ACTION TEST_CASE_1_EXEC:
                        IF vTestCases[0].state = utTestCaseStates.RUNNING THEN
	(*Run the test case*)
	IF assertLessEqual_SINT(vTestCase1_act, vTestCase1_xp) THEN
		vTestCases[0].state := utTestCaseStates.PASSED;
		vTestCases[0].msg := 'Parameter act was less than xp and function returned TRUE -> PASS';
	ELSE
		vTestCases[0].state := utTestCaseStates.FAILED;
		vTestCases[0].msg := 'Parameter act was less than xp and function returned FALSE -> FAIL';
	END_IF
END_IF
                      
END_ACTION

ACTION TEST_CASE_2_SETUP:
                        IF vTestCases[1].state = utTestCaseStates.SETUP THEN
	(*Setup the test case information*)
	vTestCases[1].id := 2;
    vTestCases[1].desc[0] := 'RETURNS TRUE WHEN PARAMETER ACT EQUAL TO XP';
    vTestCases[1].desc[1] := 'Tests if the function returns True if the parameter act is equal to parameter xp';
	vTestCases[1].desc[2] := 'PASS IF: Return value is TRUE';
	
	(*Setup needed variables*)
	vTestCase2_act := REAL_TO_SINT(115.4);
	vTestCase2_xp := REAL_TO_SINT(115.4);
END_IF
                      
END_ACTION

ACTION TEST_CASE_2_EXEC:
                        IF vTestCases[1].state = utTestCaseStates.RUNNING THEN
	(*Run the test case*)
	IF assertLessEqual_SINT(vTestCase2_act, vTestCase2_xp) THEN
		vTestCases[1].state := utTestCaseStates.PASSED;
		vTestCases[1].msg := 'Parameter act was equal to xp and function returned TRUE -> PASS';
	ELSE
		vTestCases[1].state := utTestCaseStates.FAILED;
		vTestCases[1].msg := 'Parameter act was equal to xp and function returned FALSE -> FAIL';
	END_IF
END_IF
                      
END_ACTION

ACTION TEST_CASE_3_SETUP:
                        IF vTestCases[2].state = utTestCaseStates.SETUP THEN
	(*Setup the test case information*)
	vTestCases[2].id := 3;
    vTestCases[2].desc[0] := 'RETURNS FALSE WHEN PARAMETER ACT GREATER THAN XP';
    vTestCases[2].desc[1] := 'Tests if the function returns False if the parameter act is greater than parameter xp';
	vTestCases[2].desc[2] := 'PASS IF: Return value is FALSE';
	
	(*Setup needed variables*)
	vTestCase3_act := REAL_TO_SINT(115.4);
	vTestCase3_xp := REAL_TO_SINT(85.4);
END_IF
                      
END_ACTION

ACTION TEST_CASE_3_EXEC:
                        IF vTestCases[2].state = utTestCaseStates.RUNNING THEN
	(*Run the test case*)
	IF NOT assertLessEqual_SINT(vTestCase3_act, vTestCase3_xp) THEN
		vTestCases[2].state := utTestCaseStates.PASSED;
		vTestCases[2].msg := 'Parameter act was greater than xp and function returned FALSE -> PASS';
	ELSE
		vTestCases[2].state := utTestCaseStates.FAILED;
		vTestCases[2].msg := 'Parameter act was greater than xp and function returned TRUE -> FAIL';
	END_IF
END_IF
                      
END_ACTION
END_PROGRAM

PROGRAM test_assertLess_LDATE
  VAR
    vTestCases : ARRAY[0..20] OF utTestCase;  (* Definition of all test cases for this POU *)
    testRunner : utTestSuite;  (* Test Suite fb instance to run the tests *)
    vRunAll : BOOL;  (* Manual command to run all tests for this POU *)
    vResetAll : BOOL;  (* Manual command to reset all tests for this POU *)
    vTestCase1_act : LDATE;  (* Test data 1 of test case 1 *)
    vTestCase1_xp : LDATE;  (* Test data 2 of test case 1 *)
    vTestCase2_act : LDATE;  (* Test data 1 of test case 2 *)
    vTestCase2_xp : LDATE;  (* Test data 2 of test case 2 *)
  END_VAR

                    (*Run the test cases*)
TEST_CASE_1_SETUP();
TEST_CASE_1_EXEC();

TEST_CASE_2_SETUP();
TEST_CASE_2_EXEC();

(*Instantiate the test runner*)
testRunner(
	Id := 111,
	Name := 'assertLess_LDATE',
    RunTests := GVL.RunAll OR vRunAll,
	ResetTests := GVL.ResetAll OR vResetAll,
	TestCases:=vTestCases);

(*Report the results to the collection global*)
GVL.Results[testRunner.Id] := testRunner.Summary;
                  

ACTION TEST_CASE_2_EXEC:
                        IF vTestCases[1].state = utTestCaseStates.RUNNING THEN
	(*Run the test case*)
	IF NOT assertLess_LDATE(vTestCase2_act, vTestCase2_xp) THEN
		vTestCases[1].state := utTestCaseStates.PASSED;
		vTestCases[1].msg := 'Parameter act was greater than xp and function returned FALSE -> PASS';
	ELSE
		vTestCases[1].state := utTestCaseStates.FAILED;
		vTestCases[1].msg := 'Parameter act was greater than xp and function returned TRUE -> FAIL';
	END_IF
END_IF
                      
END_ACTION

ACTION TEST_CASE_1_SETUP:
                        IF vTestCases[0].state = utTestCaseStates.SETUP THEN
	(*Setup the test case information*)
	vTestCases[0].id := 1;
	vTestCases[0].desc[0] := 'RETURNS TRUE WHEN PARAMETER ACT LESS THAN XP';
    vTestCases[0].desc[1] := 'Tests if the function returns True if the parameter act is less than parameter xp';
	vTestCases[0].desc[2] := 'PASS IF: Return value is TRUE';
	
	(*Setup needed variables*)
	vTestCase1_act := REAL_TO_LDATE(85.4);
	vTestCase1_xp := REAL_TO_LDATE(115.4);
END_IF
                      
END_ACTION

ACTION TEST_CASE_1_EXEC:
                        IF vTestCases[0].state = utTestCaseStates.RUNNING THEN
	(*Run the test case*)
	IF assertLess_LDATE(vTestCase1_act, vTestCase1_xp) THEN
		vTestCases[0].state := utTestCaseStates.PASSED;
		vTestCases[0].msg := 'Parameter act was less than xp and function returned TRUE -> PASS';
	ELSE
		vTestCases[0].state := utTestCaseStates.FAILED;
		vTestCases[0].msg := 'Parameter act was less than xp and function returned FALSE -> FAIL';
	END_IF
END_IF
                      
END_ACTION

ACTION TEST_CASE_2_SETUP:
                        IF vTestCases[1].state = utTestCaseStates.SETUP THEN
	(*Setup the test case information*)
	vTestCases[1].id := 2;
    vTestCases[1].desc[0] := 'RETURNS FALSE WHEN PARAMETER ACT GREATER THAN XP';
    vTestCases[1].desc[1] := 'Tests if the function returns False if the parameter act is greater than parameter xp';
	vTestCases[1].desc[2] := 'PASS IF: Return value is FALSE';
	
	(*Setup needed variables*)
	vTestCase2_act := REAL_TO_LDATE(115.4);
	vTestCase2_xp := REAL_TO_LDATE(85.4);
END_IF
                      
END_ACTION
END_PROGRAM

PROGRAM test_assertLess_ULINT
  VAR
    vTestCases : ARRAY[0..20] OF utTestCase;  (* Definition of all test cases for this POU *)
    testRunner : utTestSuite;  (* Test Suite fb instance to run the tests *)
    vRunAll : BOOL;  (* Manual command to run all tests for this POU *)
    vResetAll : BOOL;  (* Manual command to reset all tests for this POU *)
    vTestCase1_act : ULINT;  (* Test data 1 of test case 1 *)
    vTestCase1_xp : ULINT;  (* Test data 2 of test case 1 *)
    vTestCase2_act : ULINT;  (* Test data 1 of test case 2 *)
    vTestCase2_xp : ULINT;  (* Test data 2 of test case 2 *)
  END_VAR

                    (*Run the test cases*)
TEST_CASE_1_SETUP();
TEST_CASE_1_EXEC();

TEST_CASE_2_SETUP();
TEST_CASE_2_EXEC();

(*Instantiate the test runner*)
testRunner(
	Id := 105,
	Name := 'assertLess_ULINT',
    RunTests := GVL.RunAll OR vRunAll,
	ResetTests := GVL.ResetAll OR vResetAll,
	TestCases:=vTestCases);

(*Report the results to the collection global*)
GVL.Results[testRunner.Id] := testRunner.Summary;
                  

ACTION TEST_CASE_1_SETUP:
                        IF vTestCases[0].state = utTestCaseStates.SETUP THEN
	(*Setup the test case information*)
	vTestCases[0].id := 1;
	vTestCases[0].desc[0] := 'RETURNS TRUE WHEN PARAMETER ACT LESS THAN XP';
    vTestCases[0].desc[1] := 'Tests if the function returns True if the parameter act is less than parameter xp';
	vTestCases[0].desc[2] := 'PASS IF: Return value is TRUE';
	
	(*Setup needed variables*)
	vTestCase1_act := REAL_TO_ULINT(85.4);
	vTestCase1_xp := REAL_TO_ULINT(115.4);
END_IF
                      
END_ACTION

ACTION TEST_CASE_1_EXEC:
                        IF vTestCases[0].state = utTestCaseStates.RUNNING THEN
	(*Run the test case*)
	IF assertLess_ULINT(vTestCase1_act, vTestCase1_xp) THEN
		vTestCases[0].state := utTestCaseStates.PASSED;
		vTestCases[0].msg := 'Parameter act was less than xp and function returned TRUE -> PASS';
	ELSE
		vTestCases[0].state := utTestCaseStates.FAILED;
		vTestCases[0].msg := 'Parameter act was less than xp and function returned FALSE -> FAIL';
	END_IF
END_IF
                      
END_ACTION

ACTION TEST_CASE_2_SETUP:
                        IF vTestCases[1].state = utTestCaseStates.SETUP THEN
	(*Setup the test case information*)
	vTestCases[1].id := 2;
    vTestCases[1].desc[0] := 'RETURNS FALSE WHEN PARAMETER ACT GREATER THAN XP';
    vTestCases[1].desc[1] := 'Tests if the function returns False if the parameter act is greater than parameter xp';
	vTestCases[1].desc[2] := 'PASS IF: Return value is FALSE';
	
	(*Setup needed variables*)
	vTestCase2_act := REAL_TO_ULINT(115.4);
	vTestCase2_xp := REAL_TO_ULINT(85.4);
END_IF
                      
END_ACTION

ACTION TEST_CASE_2_EXEC:
                        IF vTestCases[1].state = utTestCaseStates.RUNNING THEN
	(*Run the test case*)
	IF NOT assertLess_ULINT(vTestCase2_act, vTestCase2_xp) THEN
		vTestCases[1].state := utTestCaseStates.PASSED;
		vTestCases[1].msg := 'Parameter act was greater than xp and function returned FALSE -> PASS';
	ELSE
		vTestCases[1].state := utTestCaseStates.FAILED;
		vTestCases[1].msg := 'Parameter act was greater than xp and function returned TRUE -> FAIL';
	END_IF
END_IF
                      
END_ACTION
END_PROGRAM

PROGRAM test_assertLess_REAL
  VAR
    vTestCases : ARRAY[0..20] OF utTestCase;  (* Definition of all test cases for this POU *)
    testRunner : utTestSuite;  (* Test Suite fb instance to run the tests *)
    vRunAll : BOOL;  (* Manual command to run all tests for this POU *)
    vResetAll : BOOL;  (* Manual command to reset all tests for this POU *)
    vTestCase1_act : REAL;  (* Test data 1 of test case 1 *)
    vTestCase1_xp : REAL;  (* Test data 2 of test case 1 *)
    vTestCase2_act : REAL;  (* Test data 1 of test case 2 *)
    vTestCase2_xp : REAL;  (* Test data 2 of test case 2 *)
  END_VAR

                    (*Run the test cases*)
TEST_CASE_1_SETUP();
TEST_CASE_1_EXEC();

TEST_CASE_2_SETUP();
TEST_CASE_2_EXEC();

(*Instantiate the test runner*)
testRunner(
	Id := 106,
	Name := 'assertLess_REAL',
    RunTests := GVL.RunAll OR vRunAll,
	ResetTests := GVL.ResetAll OR vResetAll,
	TestCases:=vTestCases);

(*Report the results to the collection global*)
GVL.Results[testRunner.Id] := testRunner.Summary;
                  

ACTION TEST_CASE_1_SETUP:
                        IF vTestCases[0].state = utTestCaseStates.SETUP THEN
	(*Setup the test case information*)
	vTestCases[0].id := 1;
	vTestCases[0].desc[0] := 'RETURNS TRUE WHEN PARAMETER ACT LESS THAN XP';
    vTestCases[0].desc[1] := 'Tests if the function returns True if the parameter act is less than parameter xp';
	vTestCases[0].desc[2] := 'PASS IF: Return value is TRUE';
	
	(*Setup needed variables*)
	vTestCase1_act := 85.4;
	vTestCase1_xp := 115.4;
END_IF
                      
END_ACTION

ACTION TEST_CASE_1_EXEC:
                        IF vTestCases[0].state = utTestCaseStates.RUNNING THEN
	(*Run the test case*)
	IF assertLess_REAL(vTestCase1_act, vTestCase1_xp) THEN
		vTestCases[0].state := utTestCaseStates.PASSED;
		vTestCases[0].msg := 'Parameter act was less than xp and function returned TRUE -> PASS';
	ELSE
		vTestCases[0].state := utTestCaseStates.FAILED;
		vTestCases[0].msg := 'Parameter act was less than xp and function returned FALSE -> FAIL';
	END_IF
END_IF
                      
END_ACTION

ACTION TEST_CASE_2_SETUP:
                        IF vTestCases[1].state = utTestCaseStates.SETUP THEN
	(*Setup the test case information*)
	vTestCases[1].id := 2;
    vTestCases[1].desc[0] := 'RETURNS FALSE WHEN PARAMETER ACT GREATER THAN XP';
    vTestCases[1].desc[1] := 'Tests if the function returns False if the parameter act is greater than parameter xp';
	vTestCases[1].desc[2] := 'PASS IF: Return value is FALSE';
	
	(*Setup needed variables*)
	vTestCase2_act := 115.4;
	vTestCase2_xp := 85.4;
END_IF
                      
END_ACTION

ACTION TEST_CASE_2_EXEC:
                        IF vTestCases[1].state = utTestCaseStates.RUNNING THEN
	(*Run the test case*)
	IF NOT assertLess_REAL(vTestCase2_act, vTestCase2_xp) THEN
		vTestCases[1].state := utTestCaseStates.PASSED;
		vTestCases[1].msg := 'Parameter act was greater than xp and function returned FALSE -> PASS';
	ELSE
		vTestCases[1].state := utTestCaseStates.FAILED;
		vTestCases[1].msg := 'Parameter act was greater than xp and function returned TRUE -> FAIL';
	END_IF
END_IF
                      
END_ACTION
END_PROGRAM

PROGRAM test_assertLess_TIME_OF_DAY
  VAR
    vTestCases : ARRAY[0..20] OF utTestCase;  (* Definition of all test cases for this POU *)
    testRunner : utTestSuite;  (* Test Suite fb instance to run the tests *)
    vRunAll : BOOL;  (* Manual command to run all tests for this POU *)
    vResetAll : BOOL;  (* Manual command to reset all tests for this POU *)
    vTestCase1_act : TOD;  (* Test data 1 of test case 1 *)
    vTestCase1_xp : TOD;  (* Test data 2 of test case 1 *)
    vTestCase2_act : TOD;  (* Test data 1 of test case 2 *)
    vTestCase2_xp : TOD;  (* Test data 2 of test case 2 *)
  END_VAR

                    (*Run the test cases*)
TEST_CASE_1_SETUP();
TEST_CASE_1_EXEC();

TEST_CASE_2_SETUP();
TEST_CASE_2_EXEC();

(*Instantiate the test runner*)
testRunner(
	Id := 114,
	Name := 'assertLess_TIME_OF_DAY',
    RunTests := GVL.RunAll OR vRunAll,
	ResetTests := GVL.ResetAll OR vResetAll,
	TestCases:=vTestCases);

(*Report the results to the collection global*)
GVL.Results[testRunner.Id] := testRunner.Summary;
                  

ACTION TEST_CASE_2_SETUP:
                        IF vTestCases[1].state = utTestCaseStates.SETUP THEN
	(*Setup the test case information*)
	vTestCases[1].id := 2;
    vTestCases[1].desc[0] := 'RETURNS FALSE WHEN PARAMETER ACT GREATER THAN XP';
    vTestCases[1].desc[1] := 'Tests if the function returns False if the parameter act is greater than parameter xp';
	vTestCases[1].desc[2] := 'PASS IF: Return value is FALSE';
	
	(*Setup needed variables*)
	vTestCase2_act := REAL_TO_TOD(115.4);
	vTestCase2_xp := REAL_TO_TOD(85.4);
END_IF
                      
END_ACTION

ACTION TEST_CASE_1_SETUP:
                        IF vTestCases[0].state = utTestCaseStates.SETUP THEN
	(*Setup the test case information*)
	vTestCases[0].id := 1;
	vTestCases[0].desc[0] := 'RETURNS TRUE WHEN PARAMETER ACT LESS THAN XP';
    vTestCases[0].desc[1] := 'Tests if the function returns True if the parameter act is less than parameter xp';
	vTestCases[0].desc[2] := 'PASS IF: Return value is TRUE';
	
	(*Setup needed variables*)
	vTestCase1_act := REAL_TO_TOD(85.4);
	vTestCase1_xp := REAL_TO_TOD(115.4);
END_IF
                      
END_ACTION

ACTION TEST_CASE_1_EXEC:
                        IF vTestCases[0].state = utTestCaseStates.RUNNING THEN
	(*Run the test case*)
	IF assertLess_TIME_OF_DAY(vTestCase1_act, vTestCase1_xp) THEN
		vTestCases[0].state := utTestCaseStates.PASSED;
		vTestCases[0].msg := 'Parameter act was less than xp and function returned TRUE -> PASS';
	ELSE
		vTestCases[0].state := utTestCaseStates.FAILED;
		vTestCases[0].msg := 'Parameter act was less than xp and function returned FALSE -> FAIL';
	END_IF
END_IF
                      
END_ACTION

ACTION TEST_CASE_2_EXEC:
                        IF vTestCases[1].state = utTestCaseStates.RUNNING THEN
	(*Run the test case*)
	IF NOT assertLess_TIME_OF_DAY(vTestCase2_act, vTestCase2_xp) THEN
		vTestCases[1].state := utTestCaseStates.PASSED;
		vTestCases[1].msg := 'Parameter act was greater than xp and function returned FALSE -> PASS';
	ELSE
		vTestCases[1].state := utTestCaseStates.FAILED;
		vTestCases[1].msg := 'Parameter act was greater than xp and function returned TRUE -> FAIL';
	END_IF
END_IF
                      
END_ACTION
END_PROGRAM

PROGRAM test_assertLess_LREAL
  VAR
    vTestCases : ARRAY[0..20] OF utTestCase;  (* Definition of all test cases for this POU *)
    testRunner : utTestSuite;  (* Test Suite fb instance to run the tests *)
    vRunAll : BOOL;  (* Manual command to run all tests for this POU *)
    vResetAll : BOOL;  (* Manual command to reset all tests for this POU *)
    vTestCase1_act : LREAL;  (* Test data 1 of test case 1 *)
    vTestCase1_xp : LREAL;  (* Test data 2 of test case 1 *)
    vTestCase2_act : LREAL;  (* Test data 1 of test case 2 *)
    vTestCase2_xp : LREAL;  (* Test data 2 of test case 2 *)
  END_VAR

                    (*Run the test cases*)
TEST_CASE_1_SETUP();
TEST_CASE_1_EXEC();

TEST_CASE_2_SETUP();
TEST_CASE_2_EXEC();

(*Instantiate the test runner*)
testRunner(
	Id := 107,
	Name := 'assertLess_LREAL',
    RunTests := GVL.RunAll OR vRunAll,
	ResetTests := GVL.ResetAll OR vResetAll,
	TestCases:=vTestCases);

(*Report the results to the collection global*)
GVL.Results[testRunner.Id] := testRunner.Summary;
                  

ACTION TEST_CASE_2_SETUP:
                        IF vTestCases[1].state = utTestCaseStates.SETUP THEN
	(*Setup the test case information*)
	vTestCases[1].id := 2;
    vTestCases[1].desc[0] := 'RETURNS FALSE WHEN PARAMETER ACT GREATER THAN XP';
    vTestCases[1].desc[1] := 'Tests if the function returns False if the parameter act is greater than parameter xp';
	vTestCases[1].desc[2] := 'PASS IF: Return value is FALSE';
	
	(*Setup needed variables*)
	vTestCase2_act := REAL_TO_LREAL(115.4);
	vTestCase2_xp := REAL_TO_LREAL(85.4);
END_IF
                      
END_ACTION

ACTION TEST_CASE_1_SETUP:
                        IF vTestCases[0].state = utTestCaseStates.SETUP THEN
	(*Setup the test case information*)
	vTestCases[0].id := 1;
	vTestCases[0].desc[0] := 'RETURNS TRUE WHEN PARAMETER ACT LESS THAN XP';
    vTestCases[0].desc[1] := 'Tests if the function returns True if the parameter act is less than parameter xp';
	vTestCases[0].desc[2] := 'PASS IF: Return value is TRUE';
	
	(*Setup needed variables*)
	vTestCase1_act := REAL_TO_LREAL(85.4);
	vTestCase1_xp := REAL_TO_LREAL(115.4);
END_IF
                      
END_ACTION

ACTION TEST_CASE_1_EXEC:
                        IF vTestCases[0].state = utTestCaseStates.RUNNING THEN
	(*Run the test case*)
	IF assertLess_LREAL(vTestCase1_act, vTestCase1_xp) THEN
		vTestCases[0].state := utTestCaseStates.PASSED;
		vTestCases[0].msg := 'Parameter act was less than xp and function returned TRUE -> PASS';
	ELSE
		vTestCases[0].state := utTestCaseStates.FAILED;
		vTestCases[0].msg := 'Parameter act was less than xp and function returned FALSE -> FAIL';
	END_IF
END_IF
                      
END_ACTION

ACTION TEST_CASE_2_EXEC:
                        IF vTestCases[1].state = utTestCaseStates.RUNNING THEN
	(*Run the test case*)
	IF NOT assertLess_LREAL(vTestCase2_act, vTestCase2_xp) THEN
		vTestCases[1].state := utTestCaseStates.PASSED;
		vTestCases[1].msg := 'Parameter act was greater than xp and function returned FALSE -> PASS';
	ELSE
		vTestCases[1].state := utTestCaseStates.FAILED;
		vTestCases[1].msg := 'Parameter act was greater than xp and function returned TRUE -> FAIL';
	END_IF
END_IF
                      
END_ACTION
END_PROGRAM

PROGRAM test_assertLess_BYTE
  VAR
    vTestCases : ARRAY[0..20] OF utTestCase;  (* Definition of all test cases for this POU *)
    testRunner : utTestSuite;  (* Test Suite fb instance to run the tests *)
    vRunAll : BOOL;  (* Manual command to run all tests for this POU *)
    vResetAll : BOOL;  (* Manual command to reset all tests for this POU *)
    vTestCase1_act : BYTE;  (* Test data 1 of test case 1 *)
    vTestCase1_xp : BYTE;  (* Test data 2 of test case 1 *)
    vTestCase2_act : BYTE;  (* Test data 1 of test case 2 *)
    vTestCase2_xp : BYTE;  (* Test data 2 of test case 2 *)
  END_VAR

                    (*Run the test cases*)
TEST_CASE_1_SETUP();
TEST_CASE_1_EXEC();

TEST_CASE_2_SETUP();
TEST_CASE_2_EXEC();

(*Instantiate the test runner*)
testRunner(
	Id := 94,
	Name := 'assertLess_BYTE',
    RunTests := GVL.RunAll OR vRunAll,
	ResetTests := GVL.ResetAll OR vResetAll,
	TestCases:=vTestCases);

(*Report the results to the collection global*)
GVL.Results[testRunner.Id] := testRunner.Summary;
                  

ACTION TEST_CASE_1_SETUP:
                        IF vTestCases[0].state = utTestCaseStates.SETUP THEN
	(*Setup the test case information*)
	vTestCases[0].id := 1;
	vTestCases[0].desc[0] := 'RETURNS TRUE WHEN PARAMETER ACT LESS THAN XP';
    vTestCases[0].desc[1] := 'Tests if the function returns True if the parameter act is less than parameter xp';
	vTestCases[0].desc[2] := 'PASS IF: Return value is TRUE';
	
	(*Setup needed variables*)
	vTestCase1_act := REAL_TO_BYTE(85.4);
	vTestCase1_xp := REAL_TO_BYTE(115.4);
END_IF
                      
END_ACTION

ACTION TEST_CASE_1_EXEC:
                        IF vTestCases[0].state = utTestCaseStates.RUNNING THEN
	(*Run the test case*)
	IF assertLess_BYTE(vTestCase1_act, vTestCase1_xp) THEN
		vTestCases[0].state := utTestCaseStates.PASSED;
		vTestCases[0].msg := 'Parameter act was less than xp and function returned TRUE -> PASS';
	ELSE
		vTestCases[0].state := utTestCaseStates.FAILED;
		vTestCases[0].msg := 'Parameter act was less than xp and function returned FALSE -> FAIL';
	END_IF
END_IF
                      
END_ACTION

ACTION TEST_CASE_2_SETUP:
                        IF vTestCases[1].state = utTestCaseStates.SETUP THEN
	(*Setup the test case information*)
	vTestCases[1].id := 2;
    vTestCases[1].desc[0] := 'RETURNS FALSE WHEN PARAMETER ACT GREATER THAN XP';
    vTestCases[1].desc[1] := 'Tests if the function returns False if the parameter act is greater than parameter xp';
	vTestCases[1].desc[2] := 'PASS IF: Return value is FALSE';
	
	(*Setup needed variables*)
	vTestCase2_act := REAL_TO_BYTE(115.4);
	vTestCase2_xp := REAL_TO_BYTE(85.4);
END_IF
                      
END_ACTION

ACTION TEST_CASE_2_EXEC:
                        IF vTestCases[1].state = utTestCaseStates.RUNNING THEN
	(*Run the test case*)
	IF NOT assertLess_BYTE(vTestCase2_act, vTestCase2_xp) THEN
		vTestCases[1].state := utTestCaseStates.PASSED;
		vTestCases[1].msg := 'Parameter act was greater than xp and function returned FALSE -> PASS';
	ELSE
		vTestCases[1].state := utTestCaseStates.FAILED;
		vTestCases[1].msg := 'Parameter act was greater than xp and function returned TRUE -> FAIL';
	END_IF
END_IF
                      
END_ACTION
END_PROGRAM

PROGRAM test_assertLess_UINT
  VAR
    vTestCases : ARRAY[0..20] OF utTestCase;  (* Definition of all test cases for this POU *)
    testRunner : utTestSuite;  (* Test Suite fb instance to run the tests *)
    vRunAll : BOOL;  (* Manual command to run all tests for this POU *)
    vResetAll : BOOL;  (* Manual command to reset all tests for this POU *)
    vTestCase1_act : UINT;  (* Test data 1 of test case 1 *)
    vTestCase1_xp : UINT;  (* Test data 2 of test case 1 *)
    vTestCase2_act : UINT;  (* Test data 1 of test case 2 *)
    vTestCase2_xp : UINT;  (* Test data 2 of test case 2 *)
  END_VAR

                    (*Run the test cases*)
TEST_CASE_1_SETUP();
TEST_CASE_1_EXEC();

TEST_CASE_2_SETUP();
TEST_CASE_2_EXEC();

(*Instantiate the test runner*)
testRunner(
	Id := 101,
	Name := 'assertLess_UINT',
    RunTests := GVL.RunAll OR vRunAll,
	ResetTests := GVL.ResetAll OR vResetAll,
	TestCases:=vTestCases);

(*Report the results to the collection global*)
GVL.Results[testRunner.Id] := testRunner.Summary;
                  

ACTION TEST_CASE_1_SETUP:
                        IF vTestCases[0].state = utTestCaseStates.SETUP THEN
	(*Setup the test case information*)
	vTestCases[0].id := 1;
	vTestCases[0].desc[0] := 'RETURNS TRUE WHEN PARAMETER ACT LESS THAN XP';
    vTestCases[0].desc[1] := 'Tests if the function returns True if the parameter act is less than parameter xp';
	vTestCases[0].desc[2] := 'PASS IF: Return value is TRUE';
	
	(*Setup needed variables*)
	vTestCase1_act := REAL_TO_UINT(85.4);
	vTestCase1_xp := REAL_TO_UINT(115.4);
END_IF
                      
END_ACTION

ACTION TEST_CASE_1_EXEC:
                        IF vTestCases[0].state = utTestCaseStates.RUNNING THEN
	(*Run the test case*)
	IF assertLess_UINT(vTestCase1_act, vTestCase1_xp) THEN
		vTestCases[0].state := utTestCaseStates.PASSED;
		vTestCases[0].msg := 'Parameter act was less than xp and function returned TRUE -> PASS';
	ELSE
		vTestCases[0].state := utTestCaseStates.FAILED;
		vTestCases[0].msg := 'Parameter act was less than xp and function returned FALSE -> FAIL';
	END_IF
END_IF
                      
END_ACTION

ACTION TEST_CASE_2_SETUP:
                        IF vTestCases[1].state = utTestCaseStates.SETUP THEN
	(*Setup the test case information*)
	vTestCases[1].id := 2;
    vTestCases[1].desc[0] := 'RETURNS FALSE WHEN PARAMETER ACT GREATER THAN XP';
    vTestCases[1].desc[1] := 'Tests if the function returns False if the parameter act is greater than parameter xp';
	vTestCases[1].desc[2] := 'PASS IF: Return value is FALSE';
	
	(*Setup needed variables*)
	vTestCase2_act := REAL_TO_UINT(115.4);
	vTestCase2_xp := REAL_TO_UINT(85.4);
END_IF
                      
END_ACTION

ACTION TEST_CASE_2_EXEC:
                        IF vTestCases[1].state = utTestCaseStates.RUNNING THEN
	(*Run the test case*)
	IF NOT assertLess_UINT(vTestCase2_act, vTestCase2_xp) THEN
		vTestCases[1].state := utTestCaseStates.PASSED;
		vTestCases[1].msg := 'Parameter act was greater than xp and function returned FALSE -> PASS';
	ELSE
		vTestCases[1].state := utTestCaseStates.FAILED;
		vTestCases[1].msg := 'Parameter act was greater than xp and function returned TRUE -> FAIL';
	END_IF
END_IF
                      
END_ACTION
END_PROGRAM

PROGRAM test_assertLess_DWORD
  VAR
    vTestCases : ARRAY[0..20] OF utTestCase;  (* Definition of all test cases for this POU *)
    testRunner : utTestSuite;  (* Test Suite fb instance to run the tests *)
    vRunAll : BOOL;  (* Manual command to run all tests for this POU *)
    vResetAll : BOOL;  (* Manual command to reset all tests for this POU *)
    vTestCase1_act : DWORD;  (* Test data 1 of test case 1 *)
    vTestCase1_xp : DWORD;  (* Test data 2 of test case 1 *)
    vTestCase2_act : DWORD;  (* Test data 1 of test case 2 *)
    vTestCase2_xp : DWORD;  (* Test data 2 of test case 2 *)
  END_VAR

                    (*Run the test cases*)
TEST_CASE_1_SETUP();
TEST_CASE_1_EXEC();

TEST_CASE_2_SETUP();
TEST_CASE_2_EXEC();

(*Instantiate the test runner*)
testRunner(
	Id := 96,
	Name := 'assertLess_DWORD',
    RunTests := GVL.RunAll OR vRunAll,
	ResetTests := GVL.ResetAll OR vResetAll,
	TestCases:=vTestCases);

(*Report the results to the collection global*)
GVL.Results[testRunner.Id] := testRunner.Summary;
                  

ACTION TEST_CASE_1_EXEC:
                        IF vTestCases[0].state = utTestCaseStates.RUNNING THEN
	(*Run the test case*)
	IF assertLess_DWORD(vTestCase1_act, vTestCase1_xp) THEN
		vTestCases[0].state := utTestCaseStates.PASSED;
		vTestCases[0].msg := 'Parameter act was less than xp and function returned TRUE -> PASS';
	ELSE
		vTestCases[0].state := utTestCaseStates.FAILED;
		vTestCases[0].msg := 'Parameter act was less than xp and function returned FALSE -> FAIL';
	END_IF
END_IF
                      
END_ACTION

ACTION TEST_CASE_2_SETUP:
                        IF vTestCases[1].state = utTestCaseStates.SETUP THEN
	(*Setup the test case information*)
	vTestCases[1].id := 2;
    vTestCases[1].desc[0] := 'RETURNS FALSE WHEN PARAMETER ACT GREATER THAN XP';
    vTestCases[1].desc[1] := 'Tests if the function returns False if the parameter act is greater than parameter xp';
	vTestCases[1].desc[2] := 'PASS IF: Return value is FALSE';
	
	(*Setup needed variables*)
	vTestCase2_act := REAL_TO_DWORD(115.4);
	vTestCase2_xp := REAL_TO_DWORD(85.4);
END_IF
                      
END_ACTION

ACTION TEST_CASE_2_EXEC:
                        IF vTestCases[1].state = utTestCaseStates.RUNNING THEN
	(*Run the test case*)
	IF NOT assertLess_DWORD(vTestCase2_act, vTestCase2_xp) THEN
		vTestCases[1].state := utTestCaseStates.PASSED;
		vTestCases[1].msg := 'Parameter act was greater than xp and function returned FALSE -> PASS';
	ELSE
		vTestCases[1].state := utTestCaseStates.FAILED;
		vTestCases[1].msg := 'Parameter act was greater than xp and function returned TRUE -> FAIL';
	END_IF
END_IF
                      
END_ACTION

ACTION TEST_CASE_1_SETUP:
                        IF vTestCases[0].state = utTestCaseStates.SETUP THEN
	(*Setup the test case information*)
	vTestCases[0].id := 1;
	vTestCases[0].desc[0] := 'RETURNS TRUE WHEN PARAMETER ACT LESS THAN XP';
    vTestCases[0].desc[1] := 'Tests if the function returns True if the parameter act is less than parameter xp';
	vTestCases[0].desc[2] := 'PASS IF: Return value is TRUE';
	
	(*Setup needed variables*)
	vTestCase1_act := REAL_TO_DWORD(85.4);
	vTestCase1_xp := REAL_TO_DWORD(115.4);
END_IF
                      
END_ACTION
END_PROGRAM

PROGRAM test_assertLess_UDINT
  VAR
    vTestCases : ARRAY[0..20] OF utTestCase;  (* Definition of all test cases for this POU *)
    testRunner : utTestSuite;  (* Test Suite fb instance to run the tests *)
    vRunAll : BOOL;  (* Manual command to run all tests for this POU *)
    vResetAll : BOOL;  (* Manual command to reset all tests for this POU *)
    vTestCase1_act : UDINT;  (* Test data 1 of test case 1 *)
    vTestCase1_xp : UDINT;  (* Test data 2 of test case 1 *)
    vTestCase2_act : UDINT;  (* Test data 1 of test case 2 *)
    vTestCase2_xp : UDINT;  (* Test data 2 of test case 2 *)
  END_VAR

                    (*Run the test cases*)
TEST_CASE_1_SETUP();
TEST_CASE_1_EXEC();

TEST_CASE_2_SETUP();
TEST_CASE_2_EXEC();

(*Instantiate the test runner*)
testRunner(
	Id := 103,
	Name := 'assertLess_UDINT',
    RunTests := GVL.RunAll OR vRunAll,
	ResetTests := GVL.ResetAll OR vResetAll,
	TestCases:=vTestCases);

(*Report the results to the collection global*)
GVL.Results[testRunner.Id] := testRunner.Summary;
                  

ACTION TEST_CASE_1_EXEC:
                        IF vTestCases[0].state = utTestCaseStates.RUNNING THEN
	(*Run the test case*)
	IF assertLess_UDINT(vTestCase1_act, vTestCase1_xp) THEN
		vTestCases[0].state := utTestCaseStates.PASSED;
		vTestCases[0].msg := 'Parameter act was less than xp and function returned TRUE -> PASS';
	ELSE
		vTestCases[0].state := utTestCaseStates.FAILED;
		vTestCases[0].msg := 'Parameter act was less than xp and function returned FALSE -> FAIL';
	END_IF
END_IF
                      
END_ACTION

ACTION TEST_CASE_2_SETUP:
                        IF vTestCases[1].state = utTestCaseStates.SETUP THEN
	(*Setup the test case information*)
	vTestCases[1].id := 2;
    vTestCases[1].desc[0] := 'RETURNS FALSE WHEN PARAMETER ACT GREATER THAN XP';
    vTestCases[1].desc[1] := 'Tests if the function returns False if the parameter act is greater than parameter xp';
	vTestCases[1].desc[2] := 'PASS IF: Return value is FALSE';
	
	(*Setup needed variables*)
	vTestCase2_act := REAL_TO_UDINT(115.4);
	vTestCase2_xp := REAL_TO_UDINT(85.4);
END_IF
                      
END_ACTION

ACTION TEST_CASE_2_EXEC:
                        IF vTestCases[1].state = utTestCaseStates.RUNNING THEN
	(*Run the test case*)
	IF NOT assertLess_UDINT(vTestCase2_act, vTestCase2_xp) THEN
		vTestCases[1].state := utTestCaseStates.PASSED;
		vTestCases[1].msg := 'Parameter act was greater than xp and function returned FALSE -> PASS';
	ELSE
		vTestCases[1].state := utTestCaseStates.FAILED;
		vTestCases[1].msg := 'Parameter act was greater than xp and function returned TRUE -> FAIL';
	END_IF
END_IF
                      
END_ACTION

ACTION TEST_CASE_1_SETUP:
                        IF vTestCases[0].state = utTestCaseStates.SETUP THEN
	(*Setup the test case information*)
	vTestCases[0].id := 1;
	vTestCases[0].desc[0] := 'RETURNS TRUE WHEN PARAMETER ACT LESS THAN XP';
    vTestCases[0].desc[1] := 'Tests if the function returns True if the parameter act is less than parameter xp';
	vTestCases[0].desc[2] := 'PASS IF: Return value is TRUE';
	
	(*Setup needed variables*)
	vTestCase1_act := REAL_TO_UDINT(85.4);
	vTestCase1_xp := REAL_TO_UDINT(115.4);
END_IF
                      
END_ACTION
END_PROGRAM

PROGRAM test_assertLess_LTIME_OF_DAY
  VAR
    vTestCases : ARRAY[0..20] OF utTestCase;  (* Definition of all test cases for this POU *)
    testRunner : utTestSuite;  (* Test Suite fb instance to run the tests *)
    vRunAll : BOOL;  (* Manual command to run all tests for this POU *)
    vResetAll : BOOL;  (* Manual command to reset all tests for this POU *)
    vTestCase1_act : LTIME_OF_DAY;  (* Test data 1 of test case 1 *)
    vTestCase1_xp : LTIME_OF_DAY;  (* Test data 2 of test case 1 *)
    vTestCase2_act : LTIME_OF_DAY;  (* Test data 1 of test case 2 *)
    vTestCase2_xp : LTIME_OF_DAY;  (* Test data 2 of test case 2 *)
  END_VAR

                    (*Run the test cases*)
TEST_CASE_1_SETUP();
TEST_CASE_1_EXEC();

TEST_CASE_2_SETUP();
TEST_CASE_2_EXEC();

(*Instantiate the test runner*)
testRunner(
	Id := 115,
	Name := 'assertLess_LTIME_OF_DAY',
    RunTests := GVL.RunAll OR vRunAll,
	ResetTests := GVL.ResetAll OR vResetAll,
	TestCases:=vTestCases);

(*Report the results to the collection global*)
GVL.Results[testRunner.Id] := testRunner.Summary;
                  

ACTION TEST_CASE_1_SETUP:
                        IF vTestCases[0].state = utTestCaseStates.SETUP THEN
	(*Setup the test case information*)
	vTestCases[0].id := 1;
	vTestCases[0].desc[0] := 'RETURNS TRUE WHEN PARAMETER ACT LESS THAN XP';
    vTestCases[0].desc[1] := 'Tests if the function returns True if the parameter act is less than parameter xp';
	vTestCases[0].desc[2] := 'PASS IF: Return value is TRUE';
	
	(*Setup needed variables*)
	vTestCase1_act := REAL_TO_LTOD(85.4);
	vTestCase1_xp := REAL_TO_LTOD(115.4);
END_IF
                      
END_ACTION

ACTION TEST_CASE_1_EXEC:
                        IF vTestCases[0].state = utTestCaseStates.RUNNING THEN
	(*Run the test case*)
	IF assertLess_LTIME_OF_DAY(vTestCase1_act, vTestCase1_xp) THEN
		vTestCases[0].state := utTestCaseStates.PASSED;
		vTestCases[0].msg := 'Parameter act was less than xp and function returned TRUE -> PASS';
	ELSE
		vTestCases[0].state := utTestCaseStates.FAILED;
		vTestCases[0].msg := 'Parameter act was less than xp and function returned FALSE -> FAIL';
	END_IF
END_IF
                      
END_ACTION

ACTION TEST_CASE_2_SETUP:
                        IF vTestCases[1].state = utTestCaseStates.SETUP THEN
	(*Setup the test case information*)
	vTestCases[1].id := 2;
    vTestCases[1].desc[0] := 'RETURNS FALSE WHEN PARAMETER ACT GREATER THAN XP';
    vTestCases[1].desc[1] := 'Tests if the function returns False if the parameter act is greater than parameter xp';
	vTestCases[1].desc[2] := 'PASS IF: Return value is FALSE';
	
	(*Setup needed variables*)
	vTestCase2_act := REAL_TO_LTOD(115.4);
	vTestCase2_xp := REAL_TO_LTOD(85.4);
END_IF
                      
END_ACTION

ACTION TEST_CASE_2_EXEC:
                        IF vTestCases[1].state = utTestCaseStates.RUNNING THEN
	(*Run the test case*)
	IF NOT assertLess_LTIME_OF_DAY(vTestCase2_act, vTestCase2_xp) THEN
		vTestCases[1].state := utTestCaseStates.PASSED;
		vTestCases[1].msg := 'Parameter act was greater than xp and function returned FALSE -> PASS';
	ELSE
		vTestCases[1].state := utTestCaseStates.FAILED;
		vTestCases[1].msg := 'Parameter act was greater than xp and function returned TRUE -> FAIL';
	END_IF
END_IF
                      
END_ACTION
END_PROGRAM

PROGRAM test_assertLess_TIME
  VAR
    vTestCases : ARRAY[0..20] OF utTestCase;  (* Definition of all test cases for this POU *)
    testRunner : utTestSuite;  (* Test Suite fb instance to run the tests *)
    vRunAll : BOOL;  (* Manual command to run all tests for this POU *)
    vResetAll : BOOL;  (* Manual command to reset all tests for this POU *)
    vTestCase1_act : TIME;  (* Test data 1 of test case 1 *)
    vTestCase1_xp : TIME;  (* Test data 2 of test case 1 *)
    vTestCase2_act : TIME;  (* Test data 1 of test case 2 *)
    vTestCase2_xp : TIME;  (* Test data 2 of test case 2 *)
  END_VAR

                    (*Run the test cases*)
TEST_CASE_1_SETUP();
TEST_CASE_1_EXEC();

TEST_CASE_2_SETUP();
TEST_CASE_2_EXEC();

(*Instantiate the test runner*)
testRunner(
	Id := 108,
	Name := 'assertLess_TIME',
    RunTests := GVL.RunAll OR vRunAll,
	ResetTests := GVL.ResetAll OR vResetAll,
	TestCases:=vTestCases);

(*Report the results to the collection global*)
GVL.Results[testRunner.Id] := testRunner.Summary;
                  

ACTION TEST_CASE_1_SETUP:
                        IF vTestCases[0].state = utTestCaseStates.SETUP THEN
	(*Setup the test case information*)
	vTestCases[0].id := 1;
	vTestCases[0].desc[0] := 'RETURNS TRUE WHEN PARAMETER ACT LESS THAN XP';
    vTestCases[0].desc[1] := 'Tests if the function returns True if the parameter act is less than parameter xp';
	vTestCases[0].desc[2] := 'PASS IF: Return value is TRUE';
	
	(*Setup needed variables*)
	vTestCase1_act := REAL_TO_TIME(85.4);
	vTestCase1_xp := REAL_TO_TIME(115.4);
END_IF
                      
END_ACTION

ACTION TEST_CASE_1_EXEC:
                        IF vTestCases[0].state = utTestCaseStates.RUNNING THEN
	(*Run the test case*)
	IF assertLess_TIME(vTestCase1_act, vTestCase1_xp) THEN
		vTestCases[0].state := utTestCaseStates.PASSED;
		vTestCases[0].msg := 'Parameter act was less than xp and function returned TRUE -> PASS';
	ELSE
		vTestCases[0].state := utTestCaseStates.FAILED;
		vTestCases[0].msg := 'Parameter act was less than xp and function returned FALSE -> FAIL';
	END_IF
END_IF
                      
END_ACTION

ACTION TEST_CASE_2_SETUP:
                        IF vTestCases[1].state = utTestCaseStates.SETUP THEN
	(*Setup the test case information*)
	vTestCases[1].id := 2;
    vTestCases[1].desc[0] := 'RETURNS FALSE WHEN PARAMETER ACT GREATER THAN XP';
    vTestCases[1].desc[1] := 'Tests if the function returns False if the parameter act is greater than parameter xp';
	vTestCases[1].desc[2] := 'PASS IF: Return value is FALSE';
	
	(*Setup needed variables*)
	vTestCase2_act := REAL_TO_TIME(115.4);
	vTestCase2_xp := REAL_TO_TIME(85.4);
END_IF
                      
END_ACTION

ACTION TEST_CASE_2_EXEC:
                        IF vTestCases[1].state = utTestCaseStates.RUNNING THEN
	(*Run the test case*)
	IF NOT assertLess_TIME(vTestCase2_act, vTestCase2_xp) THEN
		vTestCases[1].state := utTestCaseStates.PASSED;
		vTestCases[1].msg := 'Parameter act was greater than xp and function returned FALSE -> PASS';
	ELSE
		vTestCases[1].state := utTestCaseStates.FAILED;
		vTestCases[1].msg := 'Parameter act was greater than xp and function returned TRUE -> FAIL';
	END_IF
END_IF
                      
END_ACTION
END_PROGRAM

PROGRAM test_assertGreater_REAL
  VAR
    vTestCases : ARRAY[0..20] OF utTestCase;  (* Definition of all test cases for this POU *)
    testRunner : utTestSuite;  (* Test Suite fb instance to run the tests *)
    vRunAll : BOOL;  (* Manual command to run all tests for this POU *)
    vResetAll : BOOL;  (* Manual command to reset all tests for this POU *)
    vTestCase1_act : REAL;  (* Test data 1 of test case 1 *)
    vTestCase1_xp : REAL;  (* Test data 2 of test case 1 *)
    vTestCase2_act : REAL;  (* Test data 1 of test case 2 *)
    vTestCase2_xp : REAL;  (* Test data 2 of test case 2 *)
  END_VAR

                    (*Run the test cases*)
TEST_CASE_1_SETUP();
TEST_CASE_1_EXEC();

TEST_CASE_2_SETUP();
TEST_CASE_2_EXEC();

(*Instantiate the test runner*)
testRunner(
	Id := 62,
	Name := 'assertGreater_REAL',
    RunTests := GVL.RunAll OR vRunAll,
	ResetTests := GVL.ResetAll OR vResetAll,
	TestCases:=vTestCases);

(*Report the results to the collection global*)
GVL.Results[testRunner.Id] := testRunner.Summary;
                  

ACTION TEST_CASE_2_EXEC:
                        IF vTestCases[1].state = utTestCaseStates.RUNNING THEN
	(*Run the test case*)
	IF NOT assertGreater_REAL(vTestCase2_act, vTestCase2_xp) THEN
		vTestCases[1].state := utTestCaseStates.PASSED;
		vTestCases[1].msg := 'Parameter act was less than xp and function returned FALSE -> PASS';
	ELSE
		vTestCases[1].state := utTestCaseStates.FAILED;
		vTestCases[1].msg := 'Parameter act was less than xp and function returned TRUE -> FAIL';
	END_IF
END_IF
                      
END_ACTION

ACTION TEST_CASE_1_SETUP:
                        IF vTestCases[0].state = utTestCaseStates.SETUP THEN
	(*Setup the test case information*)
	vTestCases[0].id := 1;
	vTestCases[0].desc[0] := 'RETURNS TRUE WHEN PARAMETER ACT GREATER THAN XP';
    vTestCases[0].desc[1] := 'Tests if the function returns True if the parameter act is greater than parameter xp';
	vTestCases[0].desc[2] := 'PASS IF: Return value is TRUE';
	
	(*Setup needed variables*)
	vTestCase1_act := 115.4;
	vTestCase1_xp := 85.4;
END_IF
                      
END_ACTION

ACTION TEST_CASE_1_EXEC:
                        IF vTestCases[0].state = utTestCaseStates.RUNNING THEN
	(*Run the test case*)
	IF assertGreater_REAL(vTestCase1_act, vTestCase1_xp) THEN
		vTestCases[0].state := utTestCaseStates.PASSED;
		vTestCases[0].msg := 'Parameter act was greater than xp and function returned TRUE -> PASS';
	ELSE
		vTestCases[0].state := utTestCaseStates.FAILED;
		vTestCases[0].msg := 'Parameter act was greater than xp and function returned FALSE -> FAIL';
	END_IF
END_IF
                      
END_ACTION

ACTION TEST_CASE_2_SETUP:
                        IF vTestCases[1].state = utTestCaseStates.SETUP THEN
	(*Setup the test case information*)
	vTestCases[1].id := 2;
    vTestCases[1].desc[0] := 'RETURNS FALSE WHEN PARAMETER ACT LESS THAN XP';
    vTestCases[1].desc[1] := 'Tests if the function returns False if the parameter act is less than parameter xp';
	vTestCases[1].desc[2] := 'PASS IF: Return value is FALSE';
	
	(*Setup needed variables*)
	vTestCase2_act := 8.4;
	vTestCase2_xp := 85.4;
END_IF
                      
END_ACTION
END_PROGRAM

PROGRAM test_assertGreaterEqual_LDATE_AND_TIME
  VAR
    vTestCases : ARRAY[0..20] OF utTestCase;  (* Definition of all test cases for this POU *)
    testRunner : utTestSuite;  (* Test Suite fb instance to run the tests *)
    vRunAll : BOOL;  (* Manual command to run all tests for this POU *)
    vResetAll : BOOL;  (* Manual command to reset all tests for this POU *)
    vTestCase1_act : LDATE_AND_TIME;  (* Test data 1 of test case 1 *)
    vTestCase1_xp : LDATE_AND_TIME;  (* Test data 2 of test case 1 *)
    vTestCase2_act : LDATE_AND_TIME;  (* Test data 1 of test case 2 *)
    vTestCase2_xp : LDATE_AND_TIME;  (* Test data 2 of test case 2 *)
    vTestCase3_act : LDATE_AND_TIME;  (* Test data 1 of test case 3 *)
    vTestCase3_xp : LDATE_AND_TIME;  (* Test data 2 of test case 3 *)
  END_VAR

                    (*Run the test cases*)
TEST_CASE_1_SETUP();
TEST_CASE_1_EXEC();

TEST_CASE_2_SETUP();
TEST_CASE_2_EXEC();

TEST_CASE_3_SETUP();
TEST_CASE_3_EXEC();

(*Instantiate the test runner*)
testRunner(
	Id := 91,
	Name := 'assertGreaterEqual_LDATE_AND_TIME',
    RunTests := GVL.RunAll OR vRunAll,
	ResetTests := GVL.ResetAll OR vResetAll,
	TestCases:=vTestCases);

(*Report the results to the collection global*)
GVL.Results[testRunner.Id] := testRunner.Summary;
                  

ACTION TEST_CASE_1_SETUP:
                        IF vTestCases[0].state = utTestCaseStates.SETUP THEN
	(*Setup the test case information*)
	vTestCases[0].id := 1;
	vTestCases[0].desc[0] := 'RETURNS TRUE WHEN PARAMETER ACT GREATER THAN XP';
    vTestCases[0].desc[1] := 'Tests if the function returns True if the parameter act is greater than parameter xp';
	vTestCases[0].desc[2] := 'PASS IF: Return value is TRUE';
	
	(*Setup needed variables*)
	vTestCase1_act := REAL_TO_LDT(115.4);
	vTestCase1_xp := REAL_TO_LDT(85.4);
END_IF
                      
END_ACTION

ACTION TEST_CASE_1_EXEC:
                        IF vTestCases[0].state = utTestCaseStates.RUNNING THEN
	(*Run the test case*)
	IF assertGreaterEqual_LDATE_AND_TIME(vTestCase1_act, vTestCase1_xp) THEN
		vTestCases[0].state := utTestCaseStates.PASSED;
		vTestCases[0].msg := 'Parameter act was greater than xp and function returned TRUE -> PASS';
	ELSE
		vTestCases[0].state := utTestCaseStates.FAILED;
		vTestCases[0].msg := 'Parameter act was greater than xp and function returned FALSE -> FAIL';
	END_IF
END_IF
                      
END_ACTION

ACTION TEST_CASE_2_SETUP:
                        IF vTestCases[1].state = utTestCaseStates.SETUP THEN
	(*Setup the test case information*)
	vTestCases[1].id := 2;
    vTestCases[1].desc[0] := 'RETURNS TRUE WHEN PARAMETER ACT EQUAL TO XP';
    vTestCases[1].desc[1] := 'Tests if the function returns True if the parameter act is equal to parameter xp';
	vTestCases[1].desc[2] := 'PASS IF: Return value is TRUE';
	
	(*Setup needed variables*)
	vTestCase2_act := REAL_TO_LDT(115.4);
	vTestCase2_xp := REAL_TO_LDT(115.4);
END_IF
                      
END_ACTION

ACTION TEST_CASE_2_EXEC:
                        IF vTestCases[1].state = utTestCaseStates.RUNNING THEN
	(*Run the test case*)
	IF assertGreaterEqual_LDATE_AND_TIME(vTestCase2_act, vTestCase2_xp) THEN
		vTestCases[1].state := utTestCaseStates.PASSED;
		vTestCases[1].msg := 'Parameter act was equal to xp and function returned TRUE -> PASS';
	ELSE
		vTestCases[1].state := utTestCaseStates.FAILED;
		vTestCases[1].msg := 'Parameter act was equal to xp and function returned FALSE -> FAIL';
	END_IF
END_IF
                      
END_ACTION

ACTION TEST_CASE_3_SETUP:
                        IF vTestCases[2].state = utTestCaseStates.SETUP THEN
	(*Setup the test case information*)
	vTestCases[2].id := 3;
    vTestCases[2].desc[0] := 'RETURNS FALSE WHEN PARAMETER ACT LESS THAN XP';
    vTestCases[2].desc[1] := 'Tests if the function returns False if the parameter act is less than parameter xp';
	vTestCases[2].desc[2] := 'PASS IF: Return value is FALSE';
	
	(*Setup needed variables*)
	vTestCase3_act := REAL_TO_LDT(85.4);
	vTestCase3_xp := REAL_TO_LDT(115.4);
END_IF
                      
END_ACTION

ACTION TEST_CASE_3_EXEC:
                        IF vTestCases[2].state = utTestCaseStates.RUNNING THEN
	(*Run the test case*)
	IF NOT assertGreaterEqual_LDATE_AND_TIME(vTestCase3_act, vTestCase3_xp) THEN
		vTestCases[2].state := utTestCaseStates.PASSED;
		vTestCases[2].msg := 'Parameter act was less than xp and function returned FALSE -> PASS';
	ELSE
		vTestCases[2].state := utTestCaseStates.FAILED;
		vTestCases[2].msg := 'Parameter act was less than xp and function returned TRUE -> FAIL';
	END_IF
END_IF
                      
END_ACTION
END_PROGRAM

PROGRAM test_assertGreaterEqual_TIME_OF_DAY
  VAR
    vTestCases : ARRAY[0..20] OF utTestCase;  (* Definition of all test cases for this POU *)
    testRunner : utTestSuite;  (* Test Suite fb instance to run the tests *)
    vRunAll : BOOL;  (* Manual command to run all tests for this POU *)
    vResetAll : BOOL;  (* Manual command to reset all tests for this POU *)
    vTestCase1_act : TOD;  (* Test data 1 of test case 1 *)
    vTestCase1_xp : TOD;  (* Test data 2 of test case 1 *)
    vTestCase2_act : TOD;  (* Test data 1 of test case 2 *)
    vTestCase2_xp : TOD;  (* Test data 2 of test case 2 *)
    vTestCase3_act : TOD;  (* Test data 1 of test case 3 *)
    vTestCase3_xp : TOD;  (* Test data 2 of test case 3 *)
  END_VAR

                    (*Run the test cases*)
TEST_CASE_1_SETUP();
TEST_CASE_1_EXEC();

TEST_CASE_2_SETUP();
TEST_CASE_2_EXEC();

TEST_CASE_3_SETUP();
TEST_CASE_3_EXEC();

(*Instantiate the test runner*)
testRunner(
	Id := 92,
	Name := 'assertGreaterEqual_TIME_OF_DAY',
    RunTests := GVL.RunAll OR vRunAll,
	ResetTests := GVL.ResetAll OR vResetAll,
	TestCases:=vTestCases);

(*Report the results to the collection global*)
GVL.Results[testRunner.Id] := testRunner.Summary;
                  

ACTION TEST_CASE_1_SETUP:
                        IF vTestCases[0].state = utTestCaseStates.SETUP THEN
	(*Setup the test case information*)
	vTestCases[0].id := 1;
	vTestCases[0].desc[0] := 'RETURNS TRUE WHEN PARAMETER ACT GREATER THAN XP';
    vTestCases[0].desc[1] := 'Tests if the function returns True if the parameter act is greater than parameter xp';
	vTestCases[0].desc[2] := 'PASS IF: Return value is TRUE';
	
	(*Setup needed variables*)
	vTestCase1_act := REAL_TO_TOD(115.4);
	vTestCase1_xp := REAL_TO_TOD(85.4);
END_IF
                      
END_ACTION

ACTION TEST_CASE_1_EXEC:
                        IF vTestCases[0].state = utTestCaseStates.RUNNING THEN
	(*Run the test case*)
	IF assertGreaterEqual_TIME_OF_DAY(vTestCase1_act, vTestCase1_xp) THEN
		vTestCases[0].state := utTestCaseStates.PASSED;
		vTestCases[0].msg := 'Parameter act was greater than xp and function returned TRUE -> PASS';
	ELSE
		vTestCases[0].state := utTestCaseStates.FAILED;
		vTestCases[0].msg := 'Parameter act was greater than xp and function returned FALSE -> FAIL';
	END_IF
END_IF
                      
END_ACTION

ACTION TEST_CASE_2_SETUP:
                        IF vTestCases[1].state = utTestCaseStates.SETUP THEN
	(*Setup the test case information*)
	vTestCases[1].id := 2;
    vTestCases[1].desc[0] := 'RETURNS TRUE WHEN PARAMETER ACT EQUAL TO XP';
    vTestCases[1].desc[1] := 'Tests if the function returns True if the parameter act is equal to parameter xp';
	vTestCases[1].desc[2] := 'PASS IF: Return value is TRUE';
	
	(*Setup needed variables*)
	vTestCase2_act := REAL_TO_TOD(115.4);
	vTestCase2_xp := REAL_TO_TOD(115.4);
END_IF
                      
END_ACTION

ACTION TEST_CASE_2_EXEC:
                        IF vTestCases[1].state = utTestCaseStates.RUNNING THEN
	(*Run the test case*)
	IF assertGreaterEqual_TIME_OF_DAY(vTestCase2_act, vTestCase2_xp) THEN
		vTestCases[1].state := utTestCaseStates.PASSED;
		vTestCases[1].msg := 'Parameter act was equal to xp and function returned TRUE -> PASS';
	ELSE
		vTestCases[1].state := utTestCaseStates.FAILED;
		vTestCases[1].msg := 'Parameter act was equal to xp and function returned FALSE -> FAIL';
	END_IF
END_IF
                      
END_ACTION

ACTION TEST_CASE_3_SETUP:
                        IF vTestCases[2].state = utTestCaseStates.SETUP THEN
	(*Setup the test case information*)
	vTestCases[2].id := 3;
    vTestCases[2].desc[0] := 'RETURNS FALSE WHEN PARAMETER ACT LESS THAN XP';
    vTestCases[2].desc[1] := 'Tests if the function returns False if the parameter act is less than parameter xp';
	vTestCases[2].desc[2] := 'PASS IF: Return value is FALSE';
	
	(*Setup needed variables*)
	vTestCase3_act := REAL_TO_TOD(85.4);
	vTestCase3_xp := REAL_TO_TOD(115.4);
END_IF
                      
END_ACTION

ACTION TEST_CASE_3_EXEC:
                        IF vTestCases[2].state = utTestCaseStates.RUNNING THEN
	(*Run the test case*)
	IF NOT assertGreaterEqual_TIME_OF_DAY(vTestCase3_act, vTestCase3_xp) THEN
		vTestCases[2].state := utTestCaseStates.PASSED;
		vTestCases[2].msg := 'Parameter act was less than xp and function returned FALSE -> PASS';
	ELSE
		vTestCases[2].state := utTestCaseStates.FAILED;
		vTestCases[2].msg := 'Parameter act was less than xp and function returned TRUE -> FAIL';
	END_IF
END_IF
                      
END_ACTION
END_PROGRAM

PROGRAM test_assertGreater_DATE_AND_TIME
  VAR
    vTestCases : ARRAY[0..20] OF utTestCase;  (* Definition of all test cases for this POU *)
    testRunner : utTestSuite;  (* Test Suite fb instance to run the tests *)
    vRunAll : BOOL;  (* Manual command to run all tests for this POU *)
    vResetAll : BOOL;  (* Manual command to reset all tests for this POU *)
    vTestCase1_act : DT;  (* Test data 1 of test case 1 *)
    vTestCase1_xp : DT;  (* Test data 2 of test case 1 *)
    vTestCase2_act : DT;  (* Test data 1 of test case 2 *)
    vTestCase2_xp : DT;  (* Test data 2 of test case 2 *)
  END_VAR

                    (*Run the test cases*)
TEST_CASE_1_SETUP();
TEST_CASE_1_EXEC();

TEST_CASE_2_SETUP();
TEST_CASE_2_EXEC();

(*Instantiate the test runner*)
testRunner(
	Id := 68,
	Name := 'assertGreater_DATE_AND_TIME',
    RunTests := GVL.RunAll OR vRunAll,
	ResetTests := GVL.ResetAll OR vResetAll,
	TestCases:=vTestCases);

(*Report the results to the collection global*)
GVL.Results[testRunner.Id] := testRunner.Summary;
                  

ACTION TEST_CASE_1_EXEC:
                        IF vTestCases[0].state = utTestCaseStates.RUNNING THEN
	(*Run the test case*)
	IF assertGreater_DATE_AND_TIME(vTestCase1_act, vTestCase1_xp) THEN
		vTestCases[0].state := utTestCaseStates.PASSED;
		vTestCases[0].msg := 'Parameter act was greater than xp and function returned TRUE -> PASS';
	ELSE
		vTestCases[0].state := utTestCaseStates.FAILED;
		vTestCases[0].msg := 'Parameter act was greater than xp and function returned FALSE -> FAIL';
	END_IF
END_IF
                      
END_ACTION

ACTION TEST_CASE_1_SETUP:
                        IF vTestCases[0].state = utTestCaseStates.SETUP THEN
	(*Setup the test case information*)
	vTestCases[0].id := 1;
	vTestCases[0].desc[0] := 'RETURNS TRUE WHEN PARAMETER ACT GREATER THAN XP';
    vTestCases[0].desc[1] := 'Tests if the function returns True if the parameter act is greater than parameter xp';
	vTestCases[0].desc[2] := 'PASS IF: Return value is TRUE';
	
	(*Setup needed variables*)
	vTestCase1_act := REAL_TO_DT(115.4);
	vTestCase1_xp := REAL_TO_DT(85.4);
END_IF
                      
END_ACTION

ACTION TEST_CASE_2_SETUP:
                        IF vTestCases[1].state = utTestCaseStates.SETUP THEN
	(*Setup the test case information*)
	vTestCases[1].id := 2;
    vTestCases[1].desc[0] := 'RETURNS FALSE WHEN PARAMETER ACT LESS THAN XP';
    vTestCases[1].desc[1] := 'Tests if the function returns False if the parameter act is less than parameter xp';
	vTestCases[1].desc[2] := 'PASS IF: Return value is FALSE';
	
	(*Setup needed variables*)
	vTestCase2_act := REAL_TO_DT(8.4);
	vTestCase2_xp := REAL_TO_DT(85.4);
END_IF
                      
END_ACTION

ACTION TEST_CASE_2_EXEC:
                        IF vTestCases[1].state = utTestCaseStates.RUNNING THEN
	(*Run the test case*)
	IF NOT assertGreater_DATE_AND_TIME(vTestCase2_act, vTestCase2_xp) THEN
		vTestCases[1].state := utTestCaseStates.PASSED;
		vTestCases[1].msg := 'Parameter act was less than xp and function returned FALSE -> PASS';
	ELSE
		vTestCases[1].state := utTestCaseStates.FAILED;
		vTestCases[1].msg := 'Parameter act was less than xp and function returned TRUE -> FAIL';
	END_IF
END_IF
                      
END_ACTION
END_PROGRAM

PROGRAM test_assertGreaterEqual_UINT
  VAR
    vTestCases : ARRAY[0..20] OF utTestCase;  (* Definition of all test cases for this POU *)
    testRunner : utTestSuite;  (* Test Suite fb instance to run the tests *)
    vRunAll : BOOL;  (* Manual command to run all tests for this POU *)
    vResetAll : BOOL;  (* Manual command to reset all tests for this POU *)
    vTestCase1_act : UINT;  (* Test data 1 of test case 1 *)
    vTestCase1_xp : UINT;  (* Test data 2 of test case 1 *)
    vTestCase2_act : UINT;  (* Test data 1 of test case 2 *)
    vTestCase2_xp : UINT;  (* Test data 2 of test case 2 *)
    vTestCase3_act : UINT;  (* Test data 1 of test case 3 *)
    vTestCase3_xp : UINT;  (* Test data 2 of test case 3 *)
  END_VAR

                    (*Run the test cases*)
TEST_CASE_1_SETUP();
TEST_CASE_1_EXEC();

TEST_CASE_2_SETUP();
TEST_CASE_2_EXEC();

TEST_CASE_3_SETUP();
TEST_CASE_3_EXEC();

(*Instantiate the test runner*)
testRunner(
	Id := 79,
	Name := 'assertGreaterEqual_UINT',
    RunTests := GVL.RunAll OR vRunAll,
	ResetTests := GVL.ResetAll OR vResetAll,
	TestCases:=vTestCases);

(*Report the results to the collection global*)
GVL.Results[testRunner.Id] := testRunner.Summary;
                  

ACTION TEST_CASE_2_SETUP:
                        IF vTestCases[1].state = utTestCaseStates.SETUP THEN
	(*Setup the test case information*)
	vTestCases[1].id := 2;
    vTestCases[1].desc[0] := 'RETURNS TRUE WHEN PARAMETER ACT EQUAL TO XP';
    vTestCases[1].desc[1] := 'Tests if the function returns True if the parameter act is equal to parameter xp';
	vTestCases[1].desc[2] := 'PASS IF: Return value is TRUE';
	
	(*Setup needed variables*)
	vTestCase2_act := REAL_TO_UINT(115.4);
	vTestCase2_xp := REAL_TO_UINT(115.4);
END_IF
                      
END_ACTION

ACTION TEST_CASE_3_SETUP:
                        IF vTestCases[2].state = utTestCaseStates.SETUP THEN
	(*Setup the test case information*)
	vTestCases[2].id := 3;
    vTestCases[2].desc[0] := 'RETURNS FALSE WHEN PARAMETER ACT LESS THAN XP';
    vTestCases[2].desc[1] := 'Tests if the function returns False if the parameter act is less than parameter xp';
	vTestCases[2].desc[2] := 'PASS IF: Return value is FALSE';
	
	(*Setup needed variables*)
	vTestCase3_act := REAL_TO_UINT(85.4);
	vTestCase3_xp := REAL_TO_UINT(115.4);
END_IF
                      
END_ACTION

ACTION TEST_CASE_1_SETUP:
                        IF vTestCases[0].state = utTestCaseStates.SETUP THEN
	(*Setup the test case information*)
	vTestCases[0].id := 1;
	vTestCases[0].desc[0] := 'RETURNS TRUE WHEN PARAMETER ACT GREATER THAN XP';
    vTestCases[0].desc[1] := 'Tests if the function returns True if the parameter act is greater than parameter xp';
	vTestCases[0].desc[2] := 'PASS IF: Return value is TRUE';
	
	(*Setup needed variables*)
	vTestCase1_act := REAL_TO_UINT(115.4);
	vTestCase1_xp := REAL_TO_UINT(85.4);
END_IF
                      
END_ACTION

ACTION TEST_CASE_1_EXEC:
                        IF vTestCases[0].state = utTestCaseStates.RUNNING THEN
	(*Run the test case*)
	IF assertGreaterEqual_UINT(vTestCase1_act, vTestCase1_xp) THEN
		vTestCases[0].state := utTestCaseStates.PASSED;
		vTestCases[0].msg := 'Parameter act was greater than xp and function returned TRUE -> PASS';
	ELSE
		vTestCases[0].state := utTestCaseStates.FAILED;
		vTestCases[0].msg := 'Parameter act was greater than xp and function returned FALSE -> FAIL';
	END_IF
END_IF
                      
END_ACTION

ACTION TEST_CASE_2_EXEC:
                        IF vTestCases[1].state = utTestCaseStates.RUNNING THEN
	(*Run the test case*)
	IF assertGreaterEqual_UINT(vTestCase2_act, vTestCase2_xp) THEN
		vTestCases[1].state := utTestCaseStates.PASSED;
		vTestCases[1].msg := 'Parameter act was equal to xp and function returned TRUE -> PASS';
	ELSE
		vTestCases[1].state := utTestCaseStates.FAILED;
		vTestCases[1].msg := 'Parameter act was equal to xp and function returned FALSE -> FAIL';
	END_IF
END_IF
                      
END_ACTION

ACTION TEST_CASE_3_EXEC:
                        IF vTestCases[2].state = utTestCaseStates.RUNNING THEN
	(*Run the test case*)
	IF NOT assertGreaterEqual_UINT(vTestCase3_act, vTestCase3_xp) THEN
		vTestCases[2].state := utTestCaseStates.PASSED;
		vTestCases[2].msg := 'Parameter act was less than xp and function returned FALSE -> PASS';
	ELSE
		vTestCases[2].state := utTestCaseStates.FAILED;
		vTestCases[2].msg := 'Parameter act was less than xp and function returned TRUE -> FAIL';
	END_IF
END_IF
                      
END_ACTION
END_PROGRAM

PROGRAM test_assertGreaterEqual_LINT
  VAR
    vTestCases : ARRAY[0..20] OF utTestCase;  (* Definition of all test cases for this POU *)
    testRunner : utTestSuite;  (* Test Suite fb instance to run the tests *)
    vRunAll : BOOL;  (* Manual command to run all tests for this POU *)
    vResetAll : BOOL;  (* Manual command to reset all tests for this POU *)
    vTestCase1_act : LINT;  (* Test data 1 of test case 1 *)
    vTestCase1_xp : LINT;  (* Test data 2 of test case 1 *)
    vTestCase2_act : LINT;  (* Test data 1 of test case 2 *)
    vTestCase2_xp : LINT;  (* Test data 2 of test case 2 *)
    vTestCase3_act : LINT;  (* Test data 1 of test case 3 *)
    vTestCase3_xp : LINT;  (* Test data 2 of test case 3 *)
  END_VAR

                    (*Run the test cases*)
TEST_CASE_1_SETUP();
TEST_CASE_1_EXEC();

TEST_CASE_2_SETUP();
TEST_CASE_2_EXEC();

TEST_CASE_3_SETUP();
TEST_CASE_3_EXEC();

(*Instantiate the test runner*)
testRunner(
	Id := 82,
	Name := 'assertGreaterEqual_LINT',
    RunTests := GVL.RunAll OR vRunAll,
	ResetTests := GVL.ResetAll OR vResetAll,
	TestCases:=vTestCases);

(*Report the results to the collection global*)
GVL.Results[testRunner.Id] := testRunner.Summary;
                  

ACTION TEST_CASE_1_EXEC:
                        IF vTestCases[0].state = utTestCaseStates.RUNNING THEN
	(*Run the test case*)
	IF assertGreaterEqual_LINT(vTestCase1_act, vTestCase1_xp) THEN
		vTestCases[0].state := utTestCaseStates.PASSED;
		vTestCases[0].msg := 'Parameter act was greater than xp and function returned TRUE -> PASS';
	ELSE
		vTestCases[0].state := utTestCaseStates.FAILED;
		vTestCases[0].msg := 'Parameter act was greater than xp and function returned FALSE -> FAIL';
	END_IF
END_IF
                      
END_ACTION

ACTION TEST_CASE_3_EXEC:
                        IF vTestCases[2].state = utTestCaseStates.RUNNING THEN
	(*Run the test case*)
	IF NOT assertGreaterEqual_LINT(vTestCase3_act, vTestCase3_xp) THEN
		vTestCases[2].state := utTestCaseStates.PASSED;
		vTestCases[2].msg := 'Parameter act was less than xp and function returned FALSE -> PASS';
	ELSE
		vTestCases[2].state := utTestCaseStates.FAILED;
		vTestCases[2].msg := 'Parameter act was less than xp and function returned TRUE -> FAIL';
	END_IF
END_IF
                      
END_ACTION

ACTION TEST_CASE_1_SETUP:
                        IF vTestCases[0].state = utTestCaseStates.SETUP THEN
	(*Setup the test case information*)
	vTestCases[0].id := 1;
	vTestCases[0].desc[0] := 'RETURNS TRUE WHEN PARAMETER ACT GREATER THAN XP';
    vTestCases[0].desc[1] := 'Tests if the function returns True if the parameter act is greater than parameter xp';
	vTestCases[0].desc[2] := 'PASS IF: Return value is TRUE';
	
	(*Setup needed variables*)
	vTestCase1_act := REAL_TO_LINT(115.4);
	vTestCase1_xp := REAL_TO_LINT(85.4);
END_IF
                      
END_ACTION

ACTION TEST_CASE_2_SETUP:
                        IF vTestCases[1].state = utTestCaseStates.SETUP THEN
	(*Setup the test case information*)
	vTestCases[1].id := 2;
    vTestCases[1].desc[0] := 'RETURNS TRUE WHEN PARAMETER ACT EQUAL TO XP';
    vTestCases[1].desc[1] := 'Tests if the function returns True if the parameter act is equal to parameter xp';
	vTestCases[1].desc[2] := 'PASS IF: Return value is TRUE';
	
	(*Setup needed variables*)
	vTestCase2_act := REAL_TO_LINT(115.4);
	vTestCase2_xp := REAL_TO_LINT(115.4);
END_IF
                      
END_ACTION

ACTION TEST_CASE_2_EXEC:
                        IF vTestCases[1].state = utTestCaseStates.RUNNING THEN
	(*Run the test case*)
	IF assertGreaterEqual_LINT(vTestCase2_act, vTestCase2_xp) THEN
		vTestCases[1].state := utTestCaseStates.PASSED;
		vTestCases[1].msg := 'Parameter act was equal to xp and function returned TRUE -> PASS';
	ELSE
		vTestCases[1].state := utTestCaseStates.FAILED;
		vTestCases[1].msg := 'Parameter act was equal to xp and function returned FALSE -> FAIL';
	END_IF
END_IF
                      
END_ACTION

ACTION TEST_CASE_3_SETUP:
                        IF vTestCases[2].state = utTestCaseStates.SETUP THEN
	(*Setup the test case information*)
	vTestCases[2].id := 3;
    vTestCases[2].desc[0] := 'RETURNS FALSE WHEN PARAMETER ACT LESS THAN XP';
    vTestCases[2].desc[1] := 'Tests if the function returns False if the parameter act is less than parameter xp';
	vTestCases[2].desc[2] := 'PASS IF: Return value is FALSE';
	
	(*Setup needed variables*)
	vTestCase3_act := REAL_TO_LINT(85.4);
	vTestCase3_xp := REAL_TO_LINT(115.4);
END_IF
                      
END_ACTION
END_PROGRAM

PROGRAM test_assertGreaterEqual_DATE_AND_TIME
  VAR
    vTestCases : ARRAY[0..20] OF utTestCase;  (* Definition of all test cases for this POU *)
    testRunner : utTestSuite;  (* Test Suite fb instance to run the tests *)
    vRunAll : BOOL;  (* Manual command to run all tests for this POU *)
    vResetAll : BOOL;  (* Manual command to reset all tests for this POU *)
    vTestCase1_act : DT;  (* Test data 1 of test case 1 *)
    vTestCase1_xp : DT;  (* Test data 2 of test case 1 *)
    vTestCase2_act : DT;  (* Test data 1 of test case 2 *)
    vTestCase2_xp : DT;  (* Test data 2 of test case 2 *)
    vTestCase3_act : DT;  (* Test data 1 of test case 3 *)
    vTestCase3_xp : DT;  (* Test data 2 of test case 3 *)
  END_VAR

                    (*Run the test cases*)
TEST_CASE_1_SETUP();
TEST_CASE_1_EXEC();

TEST_CASE_2_SETUP();
TEST_CASE_2_EXEC();

TEST_CASE_3_SETUP();
TEST_CASE_3_EXEC();

(*Instantiate the test runner*)
testRunner(
	Id := 90,
	Name := 'assertGreaterEqual_DATE_AND_TIME',
    RunTests := GVL.RunAll OR vRunAll,
	ResetTests := GVL.ResetAll OR vResetAll,
	TestCases:=vTestCases);

(*Report the results to the collection global*)
GVL.Results[testRunner.Id] := testRunner.Summary;
                  

ACTION TEST_CASE_2_EXEC:
                        IF vTestCases[1].state = utTestCaseStates.RUNNING THEN
	(*Run the test case*)
	IF assertGreaterEqual_DATE_AND_TIME(vTestCase2_act, vTestCase2_xp) THEN
		vTestCases[1].state := utTestCaseStates.PASSED;
		vTestCases[1].msg := 'Parameter act was equal to xp and function returned TRUE -> PASS';
	ELSE
		vTestCases[1].state := utTestCaseStates.FAILED;
		vTestCases[1].msg := 'Parameter act was equal to xp and function returned FALSE -> FAIL';
	END_IF
END_IF
                      
END_ACTION

ACTION TEST_CASE_1_SETUP:
                        IF vTestCases[0].state = utTestCaseStates.SETUP THEN
	(*Setup the test case information*)
	vTestCases[0].id := 1;
	vTestCases[0].desc[0] := 'RETURNS TRUE WHEN PARAMETER ACT GREATER THAN XP';
    vTestCases[0].desc[1] := 'Tests if the function returns True if the parameter act is greater than parameter xp';
	vTestCases[0].desc[2] := 'PASS IF: Return value is TRUE';
	
	(*Setup needed variables*)
	vTestCase1_act := REAL_TO_DT(115.4);
	vTestCase1_xp := REAL_TO_DT(85.4);
END_IF
                      
END_ACTION

ACTION TEST_CASE_1_EXEC:
                        IF vTestCases[0].state = utTestCaseStates.RUNNING THEN
	(*Run the test case*)
	IF assertGreaterEqual_DATE_AND_TIME(vTestCase1_act, vTestCase1_xp) THEN
		vTestCases[0].state := utTestCaseStates.PASSED;
		vTestCases[0].msg := 'Parameter act was greater than xp and function returned TRUE -> PASS';
	ELSE
		vTestCases[0].state := utTestCaseStates.FAILED;
		vTestCases[0].msg := 'Parameter act was greater than xp and function returned FALSE -> FAIL';
	END_IF
END_IF
                      
END_ACTION

ACTION TEST_CASE_2_SETUP:
                        IF vTestCases[1].state = utTestCaseStates.SETUP THEN
	(*Setup the test case information*)
	vTestCases[1].id := 2;
    vTestCases[1].desc[0] := 'RETURNS TRUE WHEN PARAMETER ACT EQUAL TO XP';
    vTestCases[1].desc[1] := 'Tests if the function returns True if the parameter act is equal to parameter xp';
	vTestCases[1].desc[2] := 'PASS IF: Return value is TRUE';
	
	(*Setup needed variables*)
	vTestCase2_act := REAL_TO_DT(115.4);
	vTestCase2_xp := REAL_TO_DT(115.4);
END_IF
                      
END_ACTION

ACTION TEST_CASE_3_SETUP:
                        IF vTestCases[2].state = utTestCaseStates.SETUP THEN
	(*Setup the test case information*)
	vTestCases[2].id := 3;
    vTestCases[2].desc[0] := 'RETURNS FALSE WHEN PARAMETER ACT LESS THAN XP';
    vTestCases[2].desc[1] := 'Tests if the function returns False if the parameter act is less than parameter xp';
	vTestCases[2].desc[2] := 'PASS IF: Return value is FALSE';
	
	(*Setup needed variables*)
	vTestCase3_act := REAL_TO_DT(85.4);
	vTestCase3_xp := REAL_TO_DT(115.4);
END_IF
                      
END_ACTION

ACTION TEST_CASE_3_EXEC:
                        IF vTestCases[2].state = utTestCaseStates.RUNNING THEN
	(*Run the test case*)
	IF NOT assertGreaterEqual_DATE_AND_TIME(vTestCase3_act, vTestCase3_xp) THEN
		vTestCases[2].state := utTestCaseStates.PASSED;
		vTestCases[2].msg := 'Parameter act was less than xp and function returned FALSE -> PASS';
	ELSE
		vTestCases[2].state := utTestCaseStates.FAILED;
		vTestCases[2].msg := 'Parameter act was less than xp and function returned TRUE -> FAIL';
	END_IF
END_IF
                      
END_ACTION
END_PROGRAM

PROGRAM test_assertGreater_LDATE_AND_TIME
  VAR
    vTestCases : ARRAY[0..20] OF utTestCase;  (* Definition of all test cases for this POU *)
    testRunner : utTestSuite;  (* Test Suite fb instance to run the tests *)
    vRunAll : BOOL;  (* Manual command to run all tests for this POU *)
    vResetAll : BOOL;  (* Manual command to reset all tests for this POU *)
    vTestCase1_act : LDATE_AND_TIME;  (* Test data 1 of test case 1 *)
    vTestCase1_xp : LDATE_AND_TIME;  (* Test data 2 of test case 1 *)
    vTestCase2_act : LDATE_AND_TIME;  (* Test data 1 of test case 2 *)
    vTestCase2_xp : LDATE_AND_TIME;  (* Test data 2 of test case 2 *)
  END_VAR

                    (*Run the test cases*)
TEST_CASE_1_SETUP();
TEST_CASE_1_EXEC();

TEST_CASE_2_SETUP();
TEST_CASE_2_EXEC();

(*Instantiate the test runner*)
testRunner(
	Id := 69,
	Name := 'assertGreater_LDATE_AND_TIME',
    RunTests := GVL.RunAll OR vRunAll,
	ResetTests := GVL.ResetAll OR vResetAll,
	TestCases:=vTestCases);

(*Report the results to the collection global*)
GVL.Results[testRunner.Id] := testRunner.Summary;
                  

ACTION TEST_CASE_2_EXEC:
                        IF vTestCases[1].state = utTestCaseStates.RUNNING THEN
	(*Run the test case*)
	IF NOT assertGreater_LDATE_AND_TIME(vTestCase2_act, vTestCase2_xp) THEN
		vTestCases[1].state := utTestCaseStates.PASSED;
		vTestCases[1].msg := 'Parameter act was less than xp and function returned FALSE -> PASS';
	ELSE
		vTestCases[1].state := utTestCaseStates.FAILED;
		vTestCases[1].msg := 'Parameter act was less than xp and function returned TRUE -> FAIL';
	END_IF
END_IF
                      
END_ACTION

ACTION TEST_CASE_1_SETUP:
                        IF vTestCases[0].state = utTestCaseStates.SETUP THEN
	(*Setup the test case information*)
	vTestCases[0].id := 1;
	vTestCases[0].desc[0] := 'RETURNS TRUE WHEN PARAMETER ACT GREATER THAN XP';
    vTestCases[0].desc[1] := 'Tests if the function returns True if the parameter act is greater than parameter xp';
	vTestCases[0].desc[2] := 'PASS IF: Return value is TRUE';
	
	(*Setup needed variables*)
	vTestCase1_act := REAL_TO_LDT(115.4);
	vTestCase1_xp := REAL_TO_LDT(85.4);
END_IF
                      
END_ACTION

ACTION TEST_CASE_1_EXEC:
                        IF vTestCases[0].state = utTestCaseStates.RUNNING THEN
	(*Run the test case*)
	IF assertGreater_LDATE_AND_TIME(vTestCase1_act, vTestCase1_xp) THEN
		vTestCases[0].state := utTestCaseStates.PASSED;
		vTestCases[0].msg := 'Parameter act was greater than xp and function returned TRUE -> PASS';
	ELSE
		vTestCases[0].state := utTestCaseStates.FAILED;
		vTestCases[0].msg := 'Parameter act was greater than xp and function returned FALSE -> FAIL';
	END_IF
END_IF
                      
END_ACTION

ACTION TEST_CASE_2_SETUP:
                        IF vTestCases[1].state = utTestCaseStates.SETUP THEN
	(*Setup the test case information*)
	vTestCases[1].id := 2;
    vTestCases[1].desc[0] := 'RETURNS FALSE WHEN PARAMETER ACT LESS THAN XP';
    vTestCases[1].desc[1] := 'Tests if the function returns False if the parameter act is less than parameter xp';
	vTestCases[1].desc[2] := 'PASS IF: Return value is FALSE';
	
	(*Setup needed variables*)
	vTestCase2_act := REAL_TO_LDT(8.4);
	vTestCase2_xp := REAL_TO_LDT(85.4);
END_IF
                      
END_ACTION
END_PROGRAM

PROGRAM test_assertGreaterEqual_LTIME
  VAR
    vTestCases : ARRAY[0..20] OF utTestCase;  (* Definition of all test cases for this POU *)
    testRunner : utTestSuite;  (* Test Suite fb instance to run the tests *)
    vRunAll : BOOL;  (* Manual command to run all tests for this POU *)
    vResetAll : BOOL;  (* Manual command to reset all tests for this POU *)
    vTestCase1_act : LTIME;  (* Test data 1 of test case 1 *)
    vTestCase1_xp : LTIME;  (* Test data 2 of test case 1 *)
    vTestCase2_act : LTIME;  (* Test data 1 of test case 2 *)
    vTestCase2_xp : LTIME;  (* Test data 2 of test case 2 *)
    vTestCase3_act : LTIME;  (* Test data 1 of test case 3 *)
    vTestCase3_xp : LTIME;  (* Test data 2 of test case 3 *)
  END_VAR

                    (*Run the test cases*)
TEST_CASE_1_SETUP();
TEST_CASE_1_EXEC();

TEST_CASE_2_SETUP();
TEST_CASE_2_EXEC();

TEST_CASE_3_SETUP();
TEST_CASE_3_EXEC();

(*Instantiate the test runner*)
testRunner(
	Id := 87,
	Name := 'assertGreaterEqual_LTIME',
    RunTests := GVL.RunAll OR vRunAll,
	ResetTests := GVL.ResetAll OR vResetAll,
	TestCases:=vTestCases);

(*Report the results to the collection global*)
GVL.Results[testRunner.Id] := testRunner.Summary;
                  

ACTION TEST_CASE_1_SETUP:
                        IF vTestCases[0].state = utTestCaseStates.SETUP THEN
	(*Setup the test case information*)
	vTestCases[0].id := 1;
	vTestCases[0].desc[0] := 'RETURNS TRUE WHEN PARAMETER ACT GREATER THAN XP';
    vTestCases[0].desc[1] := 'Tests if the function returns True if the parameter act is greater than parameter xp';
	vTestCases[0].desc[2] := 'PASS IF: Return value is TRUE';
	
	(*Setup needed variables*)
	vTestCase1_act := REAL_TO_LTIME(115.4);
	vTestCase1_xp := REAL_TO_LTIME(85.4);
END_IF
                      
END_ACTION

ACTION TEST_CASE_1_EXEC:
                        IF vTestCases[0].state = utTestCaseStates.RUNNING THEN
	(*Run the test case*)
	IF assertGreaterEqual_LTIME(vTestCase1_act, vTestCase1_xp) THEN
		vTestCases[0].state := utTestCaseStates.PASSED;
		vTestCases[0].msg := 'Parameter act was greater than xp and function returned TRUE -> PASS';
	ELSE
		vTestCases[0].state := utTestCaseStates.FAILED;
		vTestCases[0].msg := 'Parameter act was greater than xp and function returned FALSE -> FAIL';
	END_IF
END_IF
                      
END_ACTION

ACTION TEST_CASE_2_SETUP:
                        IF vTestCases[1].state = utTestCaseStates.SETUP THEN
	(*Setup the test case information*)
	vTestCases[1].id := 2;
    vTestCases[1].desc[0] := 'RETURNS TRUE WHEN PARAMETER ACT EQUAL TO XP';
    vTestCases[1].desc[1] := 'Tests if the function returns True if the parameter act is equal to parameter xp';
	vTestCases[1].desc[2] := 'PASS IF: Return value is TRUE';
	
	(*Setup needed variables*)
	vTestCase2_act := REAL_TO_LTIME(115.4);
	vTestCase2_xp := REAL_TO_LTIME(115.4);
END_IF
                      
END_ACTION

ACTION TEST_CASE_2_EXEC:
                        IF vTestCases[1].state = utTestCaseStates.RUNNING THEN
	(*Run the test case*)
	IF assertGreaterEqual_LTIME(vTestCase2_act, vTestCase2_xp) THEN
		vTestCases[1].state := utTestCaseStates.PASSED;
		vTestCases[1].msg := 'Parameter act was equal to xp and function returned TRUE -> PASS';
	ELSE
		vTestCases[1].state := utTestCaseStates.FAILED;
		vTestCases[1].msg := 'Parameter act was equal to xp and function returned FALSE -> FAIL';
	END_IF
END_IF
                      
END_ACTION

ACTION TEST_CASE_3_SETUP:
                        IF vTestCases[2].state = utTestCaseStates.SETUP THEN
	(*Setup the test case information*)
	vTestCases[2].id := 3;
    vTestCases[2].desc[0] := 'RETURNS FALSE WHEN PARAMETER ACT LESS THAN XP';
    vTestCases[2].desc[1] := 'Tests if the function returns False if the parameter act is less than parameter xp';
	vTestCases[2].desc[2] := 'PASS IF: Return value is FALSE';
	
	(*Setup needed variables*)
	vTestCase3_act := REAL_TO_LTIME(85.4);
	vTestCase3_xp := REAL_TO_LTIME(115.4);
END_IF
                      
END_ACTION

ACTION TEST_CASE_3_EXEC:
                        IF vTestCases[2].state = utTestCaseStates.RUNNING THEN
	(*Run the test case*)
	IF NOT assertGreaterEqual_LTIME(vTestCase3_act, vTestCase3_xp) THEN
		vTestCases[2].state := utTestCaseStates.PASSED;
		vTestCases[2].msg := 'Parameter act was less than xp and function returned FALSE -> PASS';
	ELSE
		vTestCases[2].state := utTestCaseStates.FAILED;
		vTestCases[2].msg := 'Parameter act was less than xp and function returned TRUE -> FAIL';
	END_IF
END_IF
                      
END_ACTION
END_PROGRAM

PROGRAM test_assertGreater_DATE
  VAR
    vTestCases : ARRAY[0..20] OF utTestCase;  (* Definition of all test cases for this POU *)
    testRunner : utTestSuite;  (* Test Suite fb instance to run the tests *)
    vRunAll : BOOL;  (* Manual command to run all tests for this POU *)
    vResetAll : BOOL;  (* Manual command to reset all tests for this POU *)
    vTestCase1_act : DATE;  (* Test data 1 of test case 1 *)
    vTestCase1_xp : DATE;  (* Test data 2 of test case 1 *)
    vTestCase2_act : DATE;  (* Test data 1 of test case 2 *)
    vTestCase2_xp : DATE;  (* Test data 2 of test case 2 *)
  END_VAR

                    (*Run the test cases*)
TEST_CASE_1_SETUP();
TEST_CASE_1_EXEC();

TEST_CASE_2_SETUP();
TEST_CASE_2_EXEC();

(*Instantiate the test runner*)
testRunner(
	Id := 66,
	Name := 'assertGreater_DATE',
    RunTests := GVL.RunAll OR vRunAll,
	ResetTests := GVL.ResetAll OR vResetAll,
	TestCases:=vTestCases);

(*Report the results to the collection global*)
GVL.Results[testRunner.Id] := testRunner.Summary;
                  

ACTION TEST_CASE_1_SETUP:
                        IF vTestCases[0].state = utTestCaseStates.SETUP THEN
	(*Setup the test case information*)
	vTestCases[0].id := 1;
	vTestCases[0].desc[0] := 'RETURNS TRUE WHEN PARAMETER ACT GREATER THAN XP';
    vTestCases[0].desc[1] := 'Tests if the function returns True if the parameter act is greater than parameter xp';
	vTestCases[0].desc[2] := 'PASS IF: Return value is TRUE';
	
	(*Setup needed variables*)
	vTestCase1_act := REAL_TO_DATE(115.4);
	vTestCase1_xp := REAL_TO_DATE(85.4);
END_IF
                      
END_ACTION

ACTION TEST_CASE_1_EXEC:
                        IF vTestCases[0].state = utTestCaseStates.RUNNING THEN
	(*Run the test case*)
	IF assertGreater_DATE(vTestCase1_act, vTestCase1_xp) THEN
		vTestCases[0].state := utTestCaseStates.PASSED;
		vTestCases[0].msg := 'Parameter act was greater than xp and function returned TRUE -> PASS';
	ELSE
		vTestCases[0].state := utTestCaseStates.FAILED;
		vTestCases[0].msg := 'Parameter act was greater than xp and function returned FALSE -> FAIL';
	END_IF
END_IF
                      
END_ACTION

ACTION TEST_CASE_2_SETUP:
                        IF vTestCases[1].state = utTestCaseStates.SETUP THEN
	(*Setup the test case information*)
	vTestCases[1].id := 2;
    vTestCases[1].desc[0] := 'RETURNS FALSE WHEN PARAMETER ACT LESS THAN XP';
    vTestCases[1].desc[1] := 'Tests if the function returns False if the parameter act is less than parameter xp';
	vTestCases[1].desc[2] := 'PASS IF: Return value is FALSE';
	
	(*Setup needed variables*)
	vTestCase2_act := REAL_TO_DATE(8.4);
	vTestCase2_xp := REAL_TO_DATE(85.4);
END_IF
                      
END_ACTION

ACTION TEST_CASE_2_EXEC:
                        IF vTestCases[1].state = utTestCaseStates.RUNNING THEN
	(*Run the test case*)
	IF NOT assertGreater_DATE(vTestCase2_act, vTestCase2_xp) THEN
		vTestCases[1].state := utTestCaseStates.PASSED;
		vTestCases[1].msg := 'Parameter act was less than xp and function returned FALSE -> PASS';
	ELSE
		vTestCases[1].state := utTestCaseStates.FAILED;
		vTestCases[1].msg := 'Parameter act was less than xp and function returned TRUE -> FAIL';
	END_IF
END_IF
                      
END_ACTION
END_PROGRAM

PROGRAM test_assertGreaterEqual_TIME
  VAR
    vTestCases : ARRAY[0..20] OF utTestCase;  (* Definition of all test cases for this POU *)
    testRunner : utTestSuite;  (* Test Suite fb instance to run the tests *)
    vRunAll : BOOL;  (* Manual command to run all tests for this POU *)
    vResetAll : BOOL;  (* Manual command to reset all tests for this POU *)
    vTestCase1_act : TIME;  (* Test data 1 of test case 1 *)
    vTestCase1_xp : TIME;  (* Test data 2 of test case 1 *)
    vTestCase2_act : TIME;  (* Test data 1 of test case 2 *)
    vTestCase2_xp : TIME;  (* Test data 2 of test case 2 *)
    vTestCase3_act : TIME;  (* Test data 1 of test case 3 *)
    vTestCase3_xp : TIME;  (* Test data 2 of test case 3 *)
  END_VAR

                    (*Run the test cases*)
TEST_CASE_1_SETUP();
TEST_CASE_1_EXEC();

TEST_CASE_2_SETUP();
TEST_CASE_2_EXEC();

TEST_CASE_3_SETUP();
TEST_CASE_3_EXEC();

(*Instantiate the test runner*)
testRunner(
	Id := 86,
	Name := 'assertGreaterEqual_TIME',
    RunTests := GVL.RunAll OR vRunAll,
	ResetTests := GVL.ResetAll OR vResetAll,
	TestCases:=vTestCases);

(*Report the results to the collection global*)
GVL.Results[testRunner.Id] := testRunner.Summary;
                  

ACTION TEST_CASE_2_SETUP:
                        IF vTestCases[1].state = utTestCaseStates.SETUP THEN
	(*Setup the test case information*)
	vTestCases[1].id := 2;
    vTestCases[1].desc[0] := 'RETURNS TRUE WHEN PARAMETER ACT EQUAL TO XP';
    vTestCases[1].desc[1] := 'Tests if the function returns True if the parameter act is equal to parameter xp';
	vTestCases[1].desc[2] := 'PASS IF: Return value is TRUE';
	
	(*Setup needed variables*)
	vTestCase2_act := REAL_TO_TIME(115.4);
	vTestCase2_xp := REAL_TO_TIME(115.4);
END_IF
                      
END_ACTION

ACTION TEST_CASE_3_SETUP:
                        IF vTestCases[2].state = utTestCaseStates.SETUP THEN
	(*Setup the test case information*)
	vTestCases[2].id := 3;
    vTestCases[2].desc[0] := 'RETURNS FALSE WHEN PARAMETER ACT LESS THAN XP';
    vTestCases[2].desc[1] := 'Tests if the function returns False if the parameter act is less than parameter xp';
	vTestCases[2].desc[2] := 'PASS IF: Return value is FALSE';
	
	(*Setup needed variables*)
	vTestCase3_act := REAL_TO_TIME(85.4);
	vTestCase3_xp := REAL_TO_TIME(115.4);
END_IF
                      
END_ACTION

ACTION TEST_CASE_2_EXEC:
                        IF vTestCases[1].state = utTestCaseStates.RUNNING THEN
	(*Run the test case*)
	IF assertGreaterEqual_TIME(vTestCase2_act, vTestCase2_xp) THEN
		vTestCases[1].state := utTestCaseStates.PASSED;
		vTestCases[1].msg := 'Parameter act was equal to xp and function returned TRUE -> PASS';
	ELSE
		vTestCases[1].state := utTestCaseStates.FAILED;
		vTestCases[1].msg := 'Parameter act was equal to xp and function returned FALSE -> FAIL';
	END_IF
END_IF
                      
END_ACTION

ACTION TEST_CASE_1_SETUP:
                        IF vTestCases[0].state = utTestCaseStates.SETUP THEN
	(*Setup the test case information*)
	vTestCases[0].id := 1;
	vTestCases[0].desc[0] := 'RETURNS TRUE WHEN PARAMETER ACT GREATER THAN XP';
    vTestCases[0].desc[1] := 'Tests if the function returns True if the parameter act is greater than parameter xp';
	vTestCases[0].desc[2] := 'PASS IF: Return value is TRUE';
	
	(*Setup needed variables*)
	vTestCase1_act := REAL_TO_TIME(115.4);
	vTestCase1_xp := REAL_TO_TIME(85.4);
END_IF
                      
END_ACTION

ACTION TEST_CASE_1_EXEC:
                        IF vTestCases[0].state = utTestCaseStates.RUNNING THEN
	(*Run the test case*)
	IF assertGreaterEqual_TIME(vTestCase1_act, vTestCase1_xp) THEN
		vTestCases[0].state := utTestCaseStates.PASSED;
		vTestCases[0].msg := 'Parameter act was greater than xp and function returned TRUE -> PASS';
	ELSE
		vTestCases[0].state := utTestCaseStates.FAILED;
		vTestCases[0].msg := 'Parameter act was greater than xp and function returned FALSE -> FAIL';
	END_IF
END_IF
                      
END_ACTION

ACTION TEST_CASE_3_EXEC:
                        IF vTestCases[2].state = utTestCaseStates.RUNNING THEN
	(*Run the test case*)
	IF NOT assertGreaterEqual_TIME(vTestCase3_act, vTestCase3_xp) THEN
		vTestCases[2].state := utTestCaseStates.PASSED;
		vTestCases[2].msg := 'Parameter act was less than xp and function returned FALSE -> PASS';
	ELSE
		vTestCases[2].state := utTestCaseStates.FAILED;
		vTestCases[2].msg := 'Parameter act was less than xp and function returned TRUE -> FAIL';
	END_IF
END_IF
                      
END_ACTION
END_PROGRAM

PROGRAM test_assertGreaterEqual_WORD
  VAR
    vTestCases : ARRAY[0..20] OF utTestCase;  (* Definition of all test cases for this POU *)
    testRunner : utTestSuite;  (* Test Suite fb instance to run the tests *)
    vRunAll : BOOL;  (* Manual command to run all tests for this POU *)
    vResetAll : BOOL;  (* Manual command to reset all tests for this POU *)
    vTestCase1_act : WORD;  (* Test data 1 of test case 1 *)
    vTestCase1_xp : WORD;  (* Test data 2 of test case 1 *)
    vTestCase2_act : WORD;  (* Test data 1 of test case 2 *)
    vTestCase2_xp : WORD;  (* Test data 2 of test case 2 *)
    vTestCase3_act : WORD;  (* Test data 1 of test case 3 *)
    vTestCase3_xp : WORD;  (* Test data 2 of test case 3 *)
  END_VAR

                    (*Run the test cases*)
TEST_CASE_1_SETUP();
TEST_CASE_1_EXEC();

TEST_CASE_2_SETUP();
TEST_CASE_2_EXEC();

TEST_CASE_3_SETUP();
TEST_CASE_3_EXEC();

(*Instantiate the test runner*)
testRunner(
	Id := 73,
	Name := 'assertGreaterEqual_WORD',
    RunTests := GVL.RunAll OR vRunAll,
	ResetTests := GVL.ResetAll OR vResetAll,
	TestCases:=vTestCases);

(*Report the results to the collection global*)
GVL.Results[testRunner.Id] := testRunner.Summary;
                  

ACTION TEST_CASE_1_SETUP:
                        IF vTestCases[0].state = utTestCaseStates.SETUP THEN
	(*Setup the test case information*)
	vTestCases[0].id := 1;
	vTestCases[0].desc[0] := 'RETURNS TRUE WHEN PARAMETER ACT GREATER THAN XP';
    vTestCases[0].desc[1] := 'Tests if the function returns True if the parameter act is greater than parameter xp';
	vTestCases[0].desc[2] := 'PASS IF: Return value is TRUE';
	
	(*Setup needed variables*)
	vTestCase1_act := REAL_TO_WORD(115.4);
	vTestCase1_xp := REAL_TO_WORD(85.4);
END_IF
                      
END_ACTION

ACTION TEST_CASE_1_EXEC:
                        IF vTestCases[0].state = utTestCaseStates.RUNNING THEN
	(*Run the test case*)
	IF assertGreaterEqual_WORD(vTestCase1_act, vTestCase1_xp) THEN
		vTestCases[0].state := utTestCaseStates.PASSED;
		vTestCases[0].msg := 'Parameter act was greater than xp and function returned TRUE -> PASS';
	ELSE
		vTestCases[0].state := utTestCaseStates.FAILED;
		vTestCases[0].msg := 'Parameter act was greater than xp and function returned FALSE -> FAIL';
	END_IF
END_IF
                      
END_ACTION

ACTION TEST_CASE_2_SETUP:
                        IF vTestCases[1].state = utTestCaseStates.SETUP THEN
	(*Setup the test case information*)
	vTestCases[1].id := 2;
    vTestCases[1].desc[0] := 'RETURNS TRUE WHEN PARAMETER ACT EQUAL TO XP';
    vTestCases[1].desc[1] := 'Tests if the function returns True if the parameter act is equal to parameter xp';
	vTestCases[1].desc[2] := 'PASS IF: Return value is TRUE';
	
	(*Setup needed variables*)
	vTestCase2_act := REAL_TO_WORD(115.4);
	vTestCase2_xp := REAL_TO_WORD(115.4);
END_IF
                      
END_ACTION

ACTION TEST_CASE_2_EXEC:
                        IF vTestCases[1].state = utTestCaseStates.RUNNING THEN
	(*Run the test case*)
	IF assertGreaterEqual_WORD(vTestCase2_act, vTestCase2_xp) THEN
		vTestCases[1].state := utTestCaseStates.PASSED;
		vTestCases[1].msg := 'Parameter act was equal to xp and function returned TRUE -> PASS';
	ELSE
		vTestCases[1].state := utTestCaseStates.FAILED;
		vTestCases[1].msg := 'Parameter act was equal to xp and function returned FALSE -> FAIL';
	END_IF
END_IF
                      
END_ACTION

ACTION TEST_CASE_3_SETUP:
                        IF vTestCases[2].state = utTestCaseStates.SETUP THEN
	(*Setup the test case information*)
	vTestCases[2].id := 3;
    vTestCases[2].desc[0] := 'RETURNS FALSE WHEN PARAMETER ACT LESS THAN XP';
    vTestCases[2].desc[1] := 'Tests if the function returns False if the parameter act is less than parameter xp';
	vTestCases[2].desc[2] := 'PASS IF: Return value is FALSE';
	
	(*Setup needed variables*)
	vTestCase3_act := REAL_TO_WORD(85.4);
	vTestCase3_xp := REAL_TO_WORD(115.4);
END_IF
                      
END_ACTION

ACTION TEST_CASE_3_EXEC:
                        IF vTestCases[2].state = utTestCaseStates.RUNNING THEN
	(*Run the test case*)
	IF NOT assertGreaterEqual_WORD(vTestCase3_act, vTestCase3_xp) THEN
		vTestCases[2].state := utTestCaseStates.PASSED;
		vTestCases[2].msg := 'Parameter act was less than xp and function returned FALSE -> PASS';
	ELSE
		vTestCases[2].state := utTestCaseStates.FAILED;
		vTestCases[2].msg := 'Parameter act was less than xp and function returned TRUE -> FAIL';
	END_IF
END_IF
                      
END_ACTION
END_PROGRAM

PROGRAM test_assertGreaterEqual_LDATE
  VAR
    vTestCases : ARRAY[0..20] OF utTestCase;  (* Definition of all test cases for this POU *)
    testRunner : utTestSuite;  (* Test Suite fb instance to run the tests *)
    vRunAll : BOOL;  (* Manual command to run all tests for this POU *)
    vResetAll : BOOL;  (* Manual command to reset all tests for this POU *)
    vTestCase1_act : LDATE;  (* Test data 1 of test case 1 *)
    vTestCase1_xp : LDATE;  (* Test data 2 of test case 1 *)
    vTestCase2_act : LDATE;  (* Test data 1 of test case 2 *)
    vTestCase2_xp : LDATE;  (* Test data 2 of test case 2 *)
    vTestCase3_act : LDATE;  (* Test data 1 of test case 3 *)
    vTestCase3_xp : LDATE;  (* Test data 2 of test case 3 *)
  END_VAR

                    (*Run the test cases*)
TEST_CASE_1_SETUP();
TEST_CASE_1_EXEC();

TEST_CASE_2_SETUP();
TEST_CASE_2_EXEC();

TEST_CASE_3_SETUP();
TEST_CASE_3_EXEC();

(*Instantiate the test runner*)
testRunner(
	Id := 89,
	Name := 'assertGreaterEqual_LDATE',
    RunTests := GVL.RunAll OR vRunAll,
	ResetTests := GVL.ResetAll OR vResetAll,
	TestCases:=vTestCases);

(*Report the results to the collection global*)
GVL.Results[testRunner.Id] := testRunner.Summary;
                  

ACTION TEST_CASE_1_EXEC:
                        IF vTestCases[0].state = utTestCaseStates.RUNNING THEN
	(*Run the test case*)
	IF assertGreaterEqual_LDATE(vTestCase1_act, vTestCase1_xp) THEN
		vTestCases[0].state := utTestCaseStates.PASSED;
		vTestCases[0].msg := 'Parameter act was greater than xp and function returned TRUE -> PASS';
	ELSE
		vTestCases[0].state := utTestCaseStates.FAILED;
		vTestCases[0].msg := 'Parameter act was greater than xp and function returned FALSE -> FAIL';
	END_IF
END_IF
                      
END_ACTION

ACTION TEST_CASE_3_EXEC:
                        IF vTestCases[2].state = utTestCaseStates.RUNNING THEN
	(*Run the test case*)
	IF NOT assertGreaterEqual_LDATE(vTestCase3_act, vTestCase3_xp) THEN
		vTestCases[2].state := utTestCaseStates.PASSED;
		vTestCases[2].msg := 'Parameter act was less than xp and function returned FALSE -> PASS';
	ELSE
		vTestCases[2].state := utTestCaseStates.FAILED;
		vTestCases[2].msg := 'Parameter act was less than xp and function returned TRUE -> FAIL';
	END_IF
END_IF
                      
END_ACTION

ACTION TEST_CASE_2_SETUP:
                        IF vTestCases[1].state = utTestCaseStates.SETUP THEN
	(*Setup the test case information*)
	vTestCases[1].id := 2;
    vTestCases[1].desc[0] := 'RETURNS TRUE WHEN PARAMETER ACT EQUAL TO XP';
    vTestCases[1].desc[1] := 'Tests if the function returns True if the parameter act is equal to parameter xp';
	vTestCases[1].desc[2] := 'PASS IF: Return value is TRUE';
	
	(*Setup needed variables*)
	vTestCase2_act := REAL_TO_LDATE(115.4);
	vTestCase2_xp := REAL_TO_LDATE(115.4);
END_IF
                      
END_ACTION

ACTION TEST_CASE_2_EXEC:
                        IF vTestCases[1].state = utTestCaseStates.RUNNING THEN
	(*Run the test case*)
	IF assertGreaterEqual_LDATE(vTestCase2_act, vTestCase2_xp) THEN
		vTestCases[1].state := utTestCaseStates.PASSED;
		vTestCases[1].msg := 'Parameter act was equal to xp and function returned TRUE -> PASS';
	ELSE
		vTestCases[1].state := utTestCaseStates.FAILED;
		vTestCases[1].msg := 'Parameter act was equal to xp and function returned FALSE -> FAIL';
	END_IF
END_IF
                      
END_ACTION

ACTION TEST_CASE_1_SETUP:
                        IF vTestCases[0].state = utTestCaseStates.SETUP THEN
	(*Setup the test case information*)
	vTestCases[0].id := 1;
	vTestCases[0].desc[0] := 'RETURNS TRUE WHEN PARAMETER ACT GREATER THAN XP';
    vTestCases[0].desc[1] := 'Tests if the function returns True if the parameter act is greater than parameter xp';
	vTestCases[0].desc[2] := 'PASS IF: Return value is TRUE';
	
	(*Setup needed variables*)
	vTestCase1_act := REAL_TO_LDATE(115.4);
	vTestCase1_xp := REAL_TO_LDATE(85.4);
END_IF
                      
END_ACTION

ACTION TEST_CASE_3_SETUP:
                        IF vTestCases[2].state = utTestCaseStates.SETUP THEN
	(*Setup the test case information*)
	vTestCases[2].id := 3;
    vTestCases[2].desc[0] := 'RETURNS FALSE WHEN PARAMETER ACT LESS THAN XP';
    vTestCases[2].desc[1] := 'Tests if the function returns False if the parameter act is less than parameter xp';
	vTestCases[2].desc[2] := 'PASS IF: Return value is FALSE';
	
	(*Setup needed variables*)
	vTestCase3_act := REAL_TO_LDATE(85.4);
	vTestCase3_xp := REAL_TO_LDATE(115.4);
END_IF
                      
END_ACTION
END_PROGRAM

PROGRAM test_assertGreaterEqual_DINT
  VAR
    vTestCases : ARRAY[0..20] OF utTestCase;  (* Definition of all test cases for this POU *)
    testRunner : utTestSuite;  (* Test Suite fb instance to run the tests *)
    vRunAll : BOOL;  (* Manual command to run all tests for this POU *)
    vResetAll : BOOL;  (* Manual command to reset all tests for this POU *)
    vTestCase1_act : DINT;  (* Test data 1 of test case 1 *)
    vTestCase1_xp : DINT;  (* Test data 2 of test case 1 *)
    vTestCase2_act : DINT;  (* Test data 1 of test case 2 *)
    vTestCase2_xp : DINT;  (* Test data 2 of test case 2 *)
    vTestCase3_act : DINT;  (* Test data 1 of test case 3 *)
    vTestCase3_xp : DINT;  (* Test data 2 of test case 3 *)
  END_VAR

                    (*Run the test cases*)
TEST_CASE_1_SETUP();
TEST_CASE_1_EXEC();

TEST_CASE_2_SETUP();
TEST_CASE_2_EXEC();

TEST_CASE_3_SETUP();
TEST_CASE_3_EXEC();

(*Instantiate the test runner*)
testRunner(
	Id := 80,
	Name := 'assertGreaterEqual_DINT',
    RunTests := GVL.RunAll OR vRunAll,
	ResetTests := GVL.ResetAll OR vResetAll,
	TestCases:=vTestCases);

(*Report the results to the collection global*)
GVL.Results[testRunner.Id] := testRunner.Summary;
                  

ACTION TEST_CASE_1_SETUP:
                        IF vTestCases[0].state = utTestCaseStates.SETUP THEN
	(*Setup the test case information*)
	vTestCases[0].id := 1;
	vTestCases[0].desc[0] := 'RETURNS TRUE WHEN PARAMETER ACT GREATER THAN XP';
    vTestCases[0].desc[1] := 'Tests if the function returns True if the parameter act is greater than parameter xp';
	vTestCases[0].desc[2] := 'PASS IF: Return value is TRUE';
	
	(*Setup needed variables*)
	vTestCase1_act := REAL_TO_DINT(115.4);
	vTestCase1_xp := REAL_TO_DINT(85.4);
END_IF
                      
END_ACTION

ACTION TEST_CASE_1_EXEC:
                        IF vTestCases[0].state = utTestCaseStates.RUNNING THEN
	(*Run the test case*)
	IF assertGreaterEqual_DINT(vTestCase1_act, vTestCase1_xp) THEN
		vTestCases[0].state := utTestCaseStates.PASSED;
		vTestCases[0].msg := 'Parameter act was greater than xp and function returned TRUE -> PASS';
	ELSE
		vTestCases[0].state := utTestCaseStates.FAILED;
		vTestCases[0].msg := 'Parameter act was greater than xp and function returned FALSE -> FAIL';
	END_IF
END_IF
                      
END_ACTION

ACTION TEST_CASE_2_SETUP:
                        IF vTestCases[1].state = utTestCaseStates.SETUP THEN
	(*Setup the test case information*)
	vTestCases[1].id := 2;
    vTestCases[1].desc[0] := 'RETURNS TRUE WHEN PARAMETER ACT EQUAL TO XP';
    vTestCases[1].desc[1] := 'Tests if the function returns True if the parameter act is equal to parameter xp';
	vTestCases[1].desc[2] := 'PASS IF: Return value is TRUE';
	
	(*Setup needed variables*)
	vTestCase2_act := REAL_TO_DINT(115.4);
	vTestCase2_xp := REAL_TO_DINT(115.4);
END_IF
                      
END_ACTION

ACTION TEST_CASE_2_EXEC:
                        IF vTestCases[1].state = utTestCaseStates.RUNNING THEN
	(*Run the test case*)
	IF assertGreaterEqual_DINT(vTestCase2_act, vTestCase2_xp) THEN
		vTestCases[1].state := utTestCaseStates.PASSED;
		vTestCases[1].msg := 'Parameter act was equal to xp and function returned TRUE -> PASS';
	ELSE
		vTestCases[1].state := utTestCaseStates.FAILED;
		vTestCases[1].msg := 'Parameter act was equal to xp and function returned FALSE -> FAIL';
	END_IF
END_IF
                      
END_ACTION

ACTION TEST_CASE_3_SETUP:
                        IF vTestCases[2].state = utTestCaseStates.SETUP THEN
	(*Setup the test case information*)
	vTestCases[2].id := 3;
    vTestCases[2].desc[0] := 'RETURNS FALSE WHEN PARAMETER ACT LESS THAN XP';
    vTestCases[2].desc[1] := 'Tests if the function returns False if the parameter act is less than parameter xp';
	vTestCases[2].desc[2] := 'PASS IF: Return value is FALSE';
	
	(*Setup needed variables*)
	vTestCase3_act := REAL_TO_DINT(85.4);
	vTestCase3_xp := REAL_TO_DINT(115.4);
END_IF
                      
END_ACTION

ACTION TEST_CASE_3_EXEC:
                        IF vTestCases[2].state = utTestCaseStates.RUNNING THEN
	(*Run the test case*)
	IF NOT assertGreaterEqual_DINT(vTestCase3_act, vTestCase3_xp) THEN
		vTestCases[2].state := utTestCaseStates.PASSED;
		vTestCases[2].msg := 'Parameter act was less than xp and function returned FALSE -> PASS';
	ELSE
		vTestCases[2].state := utTestCaseStates.FAILED;
		vTestCases[2].msg := 'Parameter act was less than xp and function returned TRUE -> FAIL';
	END_IF
END_IF
                      
END_ACTION
END_PROGRAM

PROGRAM test_assertGreaterEqual_LWORD
  VAR
    vTestCases : ARRAY[0..20] OF utTestCase;  (* Definition of all test cases for this POU *)
    testRunner : utTestSuite;  (* Test Suite fb instance to run the tests *)
    vRunAll : BOOL;  (* Manual command to run all tests for this POU *)
    vResetAll : BOOL;  (* Manual command to reset all tests for this POU *)
    vTestCase1_act : LWORD;  (* Test data 1 of test case 1 *)
    vTestCase1_xp : LWORD;  (* Test data 2 of test case 1 *)
    vTestCase2_act : LWORD;  (* Test data 1 of test case 2 *)
    vTestCase2_xp : LWORD;  (* Test data 2 of test case 2 *)
    vTestCase3_act : LWORD;  (* Test data 1 of test case 3 *)
    vTestCase3_xp : LWORD;  (* Test data 2 of test case 3 *)
  END_VAR

                    (*Run the test cases*)
TEST_CASE_1_SETUP();
TEST_CASE_1_EXEC();

TEST_CASE_2_SETUP();
TEST_CASE_2_EXEC();

TEST_CASE_3_SETUP();
TEST_CASE_3_EXEC();

(*Instantiate the test runner*)
testRunner(
	Id := 75,
	Name := 'assertGreaterEqual_LWORD',
    RunTests := GVL.RunAll OR vRunAll,
	ResetTests := GVL.ResetAll OR vResetAll,
	TestCases:=vTestCases);

(*Report the results to the collection global*)
GVL.Results[testRunner.Id] := testRunner.Summary;
                  

ACTION TEST_CASE_1_EXEC:
                        IF vTestCases[0].state = utTestCaseStates.RUNNING THEN
	(*Run the test case*)
	IF assertGreaterEqual_LWORD(vTestCase1_act, vTestCase1_xp) THEN
		vTestCases[0].state := utTestCaseStates.PASSED;
		vTestCases[0].msg := 'Parameter act was greater than xp and function returned TRUE -> PASS';
	ELSE
		vTestCases[0].state := utTestCaseStates.FAILED;
		vTestCases[0].msg := 'Parameter act was greater than xp and function returned FALSE -> FAIL';
	END_IF
END_IF
                      
END_ACTION

ACTION TEST_CASE_3_EXEC:
                        IF vTestCases[2].state = utTestCaseStates.RUNNING THEN
	(*Run the test case*)
	IF NOT assertGreaterEqual_LWORD(vTestCase3_act, vTestCase3_xp) THEN
		vTestCases[2].state := utTestCaseStates.PASSED;
		vTestCases[2].msg := 'Parameter act was less than xp and function returned FALSE -> PASS';
	ELSE
		vTestCases[2].state := utTestCaseStates.FAILED;
		vTestCases[2].msg := 'Parameter act was less than xp and function returned TRUE -> FAIL';
	END_IF
END_IF
                      
END_ACTION

ACTION TEST_CASE_1_SETUP:
                        IF vTestCases[0].state = utTestCaseStates.SETUP THEN
	(*Setup the test case information*)
	vTestCases[0].id := 1;
	vTestCases[0].desc[0] := 'RETURNS TRUE WHEN PARAMETER ACT GREATER THAN XP';
    vTestCases[0].desc[1] := 'Tests if the function returns True if the parameter act is greater than parameter xp';
	vTestCases[0].desc[2] := 'PASS IF: Return value is TRUE';
	
	(*Setup needed variables*)
	vTestCase1_act := REAL_TO_LWORD(115.4);
	vTestCase1_xp := REAL_TO_LWORD(85.4);
END_IF
                      
